	W =  90.000 deg,	P =   0.000 deg,	R =   90.000 deg
};
P[1793]{
   GP1:
	UF : 0, UT : 6,		CONFIG : 'N U T, 0, 0, 0',
	X =  121.033  mm,	Y =   -455.775  mm,	Z =   -252.624  mm,
	W =  90.000 deg,	P =   0.000 deg,	R =   90.000 deg
};
P[1794]{
   GP1:
	UF : 0, UT : 6,		CONFIG : 'N U T, 0, 0, 0',
	X =  121.639  mm,	Y =   -456.875  mm,	Z =   -252.453  mm,
	W =  90.000 deg,	P =   0.000 deg,	R =   90.000 deg
};
P[1795]{
   GP1:
	UF : 0, UT : 6,		CONFIG : 'N U T, 0, 0, 0',
	X =  123.724  mm,	Y =   -460.404  mm,	Z =   -252.749  mm,
	W =  90.000 deg,	P =   0.000 deg,	R =   90.000 deg
};
P[1796]{
   GP1:
	UF : 0, UT : 6,		CONFIG : 'N U T, 0, 0, 0',
	X =  126.627  mm,	Y =   -465.516  mm,	Z =   -252.442  mm,
	W =  90.000 deg,	P =   0.000 deg,	R =   90.000 deg
};
P[1797]{
   GP1:
	UF : 0, UT : 6,		CONFIG : 'N U T, 0, 0, 0',
	X =  128.686  mm,	Y =   -468.983  mm,	Z =   -252.799  mm,
	W =  90.000 deg,	P =   0.000 deg,	R =   90.000 deg
};
P[1798]{
   GP1:
	UF : 0, UT : 6,		CONFIG : 'N U T, 0, 0, 0',
	X =  130.202  mm,	Y =   -471.604  mm,	Z =   -252.810  mm,
	W =  90.000 deg,	P =   0.000 deg,	R =   90.000 deg
};
P[1799]{
   GP1:
	UF : 0, UT : 6,		CONFIG : 'N U T, 0, 0, 0',
	X =  130.436  mm,	Y =   -472.132  mm,	Z =   -252.379  mm,
	W =  90.000 deg,	P =   0.000 deg,	R =   90.000 deg
};
P[1800]{
   GP1:
	UF : 0, UT : 6,		CONFIG : 'N U T, 0, 0, 0',
	X =  130.954  mm,	Y =   -472.905  mm,	Z =   -252.816  mm,
	W =  90.000 deg,	P =   0.000 deg,	R =   90.000 deg
};
P[1801]{
   GP1:
	UF : 0, UT : 6,		CONFIG : 'N U T, 0, 0, 0',
	X =  133.177  mm,	Y =   -476.831  mm,	Z =   -252.548  mm,
	W =  90.000 deg,	P =   0.000 deg,	R =   90.000 deg
};
P[1802]{
   GP1:
	UF : 0, UT : 6,		CONFIG : 'N U T, 0, 0, 0',
	X =  133.538  mm,	Y =   -477.462  mm,	Z =   -252.531  mm,
	W =  90.000 deg,	P =   0.000 deg,	R =   90.000 deg
};
P[1803]{
   GP1:
	UF : 0, UT : 6,		CONFIG : 'N U T, 0, 0, 0',
	X =  134.693  mm,	Y =   -479.414  mm,	Z =   -252.701  mm,
	W =  90.000 deg,	P =   0.000 deg,	R =   90.000 deg
};
P[1804]{
   GP1:
	UF : 0, UT : 6,		CONFIG : 'N U T, 0, 0, 0',
	X =  135.165  mm,	Y =   -480.194  mm,	Z =   -252.830  mm,
	W =  90.000 deg,	P =   0.000 deg,	R =   90.000 deg
};
P[1805]{
   GP1:
	UF : 0, UT : 6,		CONFIG : 'N U T, 0, 0, 0',
	X =  136.001  mm,	Y =   -481.750  mm,	Z =   -252.452  mm,
	W =  90.000 deg,	P =   0.000 deg,	R =   90.000 deg
};
P[1806]{
   GP1:
	UF : 0, UT : 6,		CONFIG : 'N U T, 0, 0, 0',
	X =  137.192  mm,	Y =   -483.729  mm,	Z =   -252.749  mm,
	W =  90.000 deg,	P =   0.000 deg,	R =   90.000 deg
};
P[1807]{
   GP1:
	UF : 0, UT : 6,		CONFIG : 'N U T, 0, 0, 0',
	X =  137.849  mm,	Y =   -484.896  mm,	Z =   -252.640  mm,
	W =  90.000 deg,	P =   0.000 deg,	R =   90.000 deg
};
P[1808]{
   GP1:
	UF : 0, UT : 6,		CONFIG : 'N U T, 0, 0, 0',
	X =  139.190  mm,	Y =   -487.189  mm,	Z =   -252.746  mm,
	W =  90.000 deg,	P =   0.000 deg,	R =   90.000 deg
};
P[1809]{
   GP1:
	UF : 0, UT : 6,		CONFIG : 'N U T, 0, 0, 0',
	X =  141.251  mm,	Y =   -490.781  mm,	Z =   -252.665  mm,
	W =  90.000 deg,	P =   0.000 deg,	R =   90.000 deg
};
P[1810]{
   GP1:
	UF : 0, UT : 6,		CONFIG : 'N U T, 0, 0, 0',
	X =  141.636  mm,	Y =   -491.445  mm,	Z =   -252.673  mm,
	W =  90.000 deg,	P =   0.000 deg,	R =   90.000 deg
};
P[1811]{
   GP1:
	UF : 0, UT : 6,		CONFIG : 'N U T, 0, 0, 0',
	X =  142.493  mm,	Y =   -492.972  mm,	Z =   -252.521  mm,
	W =  90.000 deg,	P =   0.000 deg,	R =   90.000 deg
};
P[1812]{
   GP1:
	UF : 0, UT : 6,		CONFIG : 'N U T, 0, 0, 0',
	X =  142.853  mm,	Y =   -493.613  mm,	Z =   -252.462  mm,
	W =  90.000 deg,	P =   0.000 deg,	R =   90.000 deg
};
P[1813]{
   GP1:
	UF : 0, UT : 6,		CONFIG : 'N U T, 0, 0, 0',
	X =  143.399  mm,	Y =   -494.516  mm,	Z =   -252.613  mm,
	W =  90.000 deg,	P =   0.000 deg,	R =   90.000 deg
};
P[1814]{
   GP1:
	UF : 0, UT : 6,		CONFIG : 'N U T, 0, 0, 0',
	X =  144.231  mm,	Y =   -495.934  mm,	Z =   -252.696  mm,
	W =  90.000 deg,	P =   0.000 deg,	R =   90.000 deg
};
P[1815]{
   GP1:
	UF : 0, UT : 6,		CONFIG : 'N U T, 0, 0, 0',
	X =  144.802  mm,	Y =   -496.952  mm,	Z =   -252.588  mm,
	W =  90.000 deg,	P =   0.000 deg,	R =   90.000 deg
};
P[1816]{
   GP1:
	UF : 0, UT : 6,		CONFIG : 'N U T, 0, 0, 0',
	X =  145.481  mm,	Y =   -498.169  mm,	Z =   -252.452  mm,
	W =  90.000 deg,	P =   0.000 deg,	R =   90.000 deg
};
P[1817]{
   GP1:
	UF : 0, UT : 6,		CONFIG : 'N U T, 0, 0, 0',
	X =  146.292  mm,	Y =   -499.476  mm,	Z =   -252.791  mm,
	W =  90.000 deg,	P =   0.000 deg,	R =   90.000 deg
};
P[1818]{
   GP1:
	UF : 0, UT : 6,		CONFIG : 'N U T, 0, 0, 0',
	X =  146.739  mm,	Y =   -500.274  mm,	Z =   -252.706  mm,
	W =  90.000 deg,	P =   0.000 deg,	R =   90.000 deg
};
P[1819]{
   GP1:
	UF : 0, UT : 6,		CONFIG : 'N U T, 0, 0, 0',
	X =  147.563  mm,	Y =   -501.701  mm,	Z =   -252.713  mm,
	W =  90.000 deg,	P =   0.000 deg,	R =   90.000 deg
};
P[1820]{
   GP1:
	UF : 0, UT : 6,		CONFIG : 'N U T, 0, 0, 0',
	X =  148.493  mm,	Y =   -503.314  mm,	Z =   -252.700  mm,
	W =  90.000 deg,	P =   0.000 deg,	R =   90.000 deg
};
P[1821]{
   GP1:
	UF : 0, UT : 6,		CONFIG : 'N U T, 0, 0, 0',
	X =  150.357  mm,	Y =   -506.621  mm,	Z =   -252.426  mm,
	W =  90.000 deg,	P =   0.000 deg,	R =   90.000 deg
};
P[1822]{
   GP1:
	UF : 0, UT : 6,		CONFIG : 'N U T, 0, 0, 0',
	X =  150.746  mm,	Y =   -507.235  mm,	Z =   -252.633  mm,
	W =  90.000 deg,	P =   0.000 deg,	R =   90.000 deg
};
P[1823]{
   GP1:
	UF : 0, UT : 6,		CONFIG : 'N U T, 0, 0, 0',
	X =  151.308  mm,	Y =   -508.160  mm,	Z =   -252.806  mm,
	W =  90.000 deg,	P =   0.000 deg,	R =   90.000 deg
};
P[1824]{
   GP1:
	UF : 0, UT : 6,		CONFIG : 'N U T, 0, 0, 0',
	X =  151.683  mm,	Y =   -508.837  mm,	Z =   -252.707  mm,
	W =  90.000 deg,	P =   0.000 deg,	R =   90.000 deg
};
P[1825]{
   GP1:
	UF : 0, UT : 6,		CONFIG : 'N U T, 0, 0, 0',
	X =  152.311  mm,	Y =   -509.929  mm,	Z =   -252.694  mm,
	W =  90.000 deg,	P =   0.000 deg,	R =   90.000 deg
};
P[1826]{
   GP1:
	UF : 0, UT : 6,		CONFIG : 'N U T, 0, 0, 0',
	X =  153.128  mm,	Y =   -511.311  mm,	Z =   -252.808  mm,
	W =  90.000 deg,	P =   0.000 deg,	R =   90.000 deg
};
P[1827]{
   GP1:
	UF : 0, UT : 6,		CONFIG : 'N U T, 0, 0, 0',
	X =  154.119  mm,	Y =   -513.068  mm,	Z =   -252.664  mm,
	W =  90.000 deg,	P =   0.000 deg,	R =   90.000 deg
};
P[1828]{
   GP1:
	UF : 0, UT : 6,		CONFIG : 'N U T, 0, 0, 0',
	X =  154.577  mm,	Y =   -513.838  mm,	Z =   -252.751  mm,
	W =  90.000 deg,	P =   0.000 deg,	R =   90.000 deg
};
P[1829]{
   GP1:
	UF : 0, UT : 6,		CONFIG : 'N U T, 0, 0, 0',
	X =  155.039  mm,	Y =   -514.717  mm,	Z =   -252.472  mm,
	W =  90.000 deg,	P =   0.000 deg,	R =   90.000 deg
};
P[1830]{
   GP1:
	UF : 0, UT : 6,		CONFIG : 'N U T, 0, 0, 0',
	X =  155.863  mm,	Y =   -516.048  mm,	Z =   -252.802  mm,
	W =  90.000 deg,	P =   0.000 deg,	R =   90.000 deg
};
P[1831]{
   GP1:
	UF : 0, UT : 6,		CONFIG : 'N U T, 0, 0, 0',
	X =  156.629  mm,	Y =   -517.370  mm,	Z =   -252.825  mm,
	W =  90.000 deg,	P =   0.000 deg,	R =   90.000 deg
};
P[1832]{
   GP1:
	UF : 0, UT : 6,		CONFIG : 'N U T, 0, 0, 0',
	X =  157.305  mm,	Y =   -518.557  mm,	Z =   -252.770  mm,
	W =  90.000 deg,	P =   0.000 deg,	R =   90.000 deg
};
P[1833]{
   GP1:
	UF : 0, UT : 6,		CONFIG : 'N U T, 0, 0, 0',
	X =  157.876  mm,	Y =   -519.576  mm,	Z =   -252.661  mm,
	W =  90.000 deg,	P =   0.000 deg,	R =   90.000 deg
};
P[1834]{
   GP1:
	UF : 0, UT : 6,		CONFIG : 'N U T, 0, 0, 0',
	X =  158.508  mm,	Y =   -520.674  mm,	Z =   -252.645  mm,
	W =  90.000 deg,	P =   0.000 deg,	R =   90.000 deg
};
P[1835]{
   GP1:
	UF : 0, UT : 6,		CONFIG : 'N U T, 0, 0, 0',
	X =  159.166  mm,	Y =   -521.778  mm,	Z =   -252.774  mm,
	W =  90.000 deg,	P =   0.000 deg,	R =   90.000 deg
};
P[1836]{
   GP1:
	UF : 0, UT : 6,		CONFIG : 'N U T, 0, 0, 0',
	X =  160.291  mm,	Y =   -523.722  mm,	Z =   -252.795  mm,
	W =  90.000 deg,	P =   0.000 deg,	R =   90.000 deg
};
P[1837]{
   GP1:
	UF : 0, UT : 6,		CONFIG : 'N U T, 0, 0, 0',
	X =  161.266  mm,	Y =   -525.519  mm,	Z =   -252.405  mm,
	W =  90.000 deg,	P =   0.000 deg,	R =   90.000 deg
};
P[1838]{
   GP1:
	UF : 0, UT : 6,		CONFIG : 'N U T, 0, 0, 0',
	X =  161.814  mm,	Y =   -526.350  mm,	Z =   -252.825  mm,
	W =  90.000 deg,	P =   0.000 deg,	R =   90.000 deg
};
P[1839]{
   GP1:
	UF : 0, UT : 6,		CONFIG : 'N U T, 0, 0, 0',
	X =  162.568  mm,	Y =   -527.699  mm,	Z =   -252.671  mm,
	W =  90.000 deg,	P =   0.000 deg,	R =   90.000 deg
};
P[1840]{
   GP1:
	UF : 0, UT : 6,		CONFIG : 'N U T, 0, 0, 0',
	X =  164.174  mm,	Y =   -530.541  mm,	Z =   -252.453  mm,
	W =  90.000 deg,	P =   0.000 deg,	R =   90.000 deg
};
P[1841]{
   GP1:
	UF : 0, UT : 6,		CONFIG : 'N U T, 0, 0, 0',
	X =  164.838  mm,	Y =   -531.586  mm,	Z =   -252.828  mm,
	W =  90.000 deg,	P =   0.000 deg,	R =   90.000 deg
};
P[1842]{
   GP1:
	UF : 0, UT : 6,		CONFIG : 'N U T, 0, 0, 0',
	X =  165.390  mm,	Y =   -532.385  mm,	Z =   -252.752  mm,
	W =  90.000 deg,	P =   0.000 deg,	R =   90.000 deg
};
P[1843]{
   GP1:
	UF : 0, UT : 6,		CONFIG : 'N U T, 0, 0, 0',
	X =  167.108  mm,	Y =   -533.626  mm,	Z =   -252.674  mm,
	W =  90.000 deg,	P =   0.000 deg,	R =   90.000 deg
};
P[1844]{
   GP1:
	UF : 0, UT : 6,		CONFIG : 'N U T, 0, 0, 0',
	X =  169.365  mm,	Y =   -533.792  mm,	Z =   -252.630  mm,
	W =  90.000 deg,	P =   0.000 deg,	R =   90.000 deg
};
P[1845]{
   GP1:
	UF : 0, UT : 6,		CONFIG : 'N U T, 0, 0, 0',
	X =  171.435  mm,	Y =   -532.869  mm,	Z =   -252.655  mm,
	W =  90.000 deg,	P =   0.000 deg,	R =   90.000 deg
};
P[1846]{
   GP1:
	UF : 0, UT : 6,		CONFIG : 'N U T, 0, 0, 0',
	X =  173.601  mm,	Y =   -531.593  mm,	Z =   -252.810  mm,
	W =  90.000 deg,	P =   0.000 deg,	R =   90.000 deg
};
P[1847]{
   GP1:
	UF : 0, UT : 6,		CONFIG : 'N U T, 0, 0, 0',
	X =  175.185  mm,	Y =   -530.681  mm,	Z =   -252.802  mm,
	W =  90.000 deg,	P =   0.000 deg,	R =   90.000 deg
};
P[1848]{
   GP1:
	UF : 0, UT : 6,		CONFIG : 'N U T, 0, 0, 0',
	X =  175.965  mm,	Y =   -530.243  mm,	Z =   -252.720  mm,
	W =  90.000 deg,	P =   0.000 deg,	R =   90.000 deg
};
P[1849]{
   GP1:
	UF : 0, UT : 6,		CONFIG : 'N U T, 0, 0, 0',
	X =  178.959  mm,	Y =   -528.516  mm,	Z =   -252.708  mm,
	W =  90.000 deg,	P =   0.000 deg,	R =   90.000 deg
};
P[1850]{
   GP1:
	UF : 0, UT : 6,		CONFIG : 'N U T, 0, 0, 0',
	X =  179.592  mm,	Y =   -528.151  mm,	Z =   -252.706  mm,
	W =  90.000 deg,	P =   0.000 deg,	R =   90.000 deg
};
P[1851]{
   GP1:
	UF : 0, UT : 6,		CONFIG : 'N U T, 0, 0, 0',
	X =  180.571  mm,	Y =   -527.618  mm,	Z =   -252.501  mm,
	W =  90.000 deg,	P =   0.000 deg,	R =   90.000 deg
};
P[1852]{
   GP1:
	UF : 0, UT : 6,		CONFIG : 'N U T, 0, 0, 0',
	X =  182.092  mm,	Y =   -526.698  mm,	Z =   -252.768  mm,
	W =  90.000 deg,	P =   0.000 deg,	R =   90.000 deg
};
P[1853]{
   GP1:
	UF : 0, UT : 6,		CONFIG : 'N U T, 0, 0, 0',
	X =  183.945  mm,	Y =   -525.646  mm,	Z =   -252.650  mm,
	W =  90.000 deg,	P =   0.000 deg,	R =   90.000 deg
};
P[1854]{
   GP1:
	UF : 0, UT : 6,		CONFIG : 'N U T, 0, 0, 0',
	X =  184.968  mm,	Y =   -525.038  mm,	Z =   -252.757  mm,
	W =  90.000 deg,	P =   0.000 deg,	R =   90.000 deg
};
P[1855]{
   GP1:
	UF : 0, UT : 6,		CONFIG : 'N U T, 0, 0, 0',
	X =  185.590  mm,	Y =   -524.689  mm,	Z =   -252.697  mm,
	W =  90.000 deg,	P =   0.000 deg,	R =   90.000 deg
};
P[1856]{
   GP1:
	UF : 0, UT : 6,		CONFIG : 'N U T, 0, 0, 0',
	X =  186.996  mm,	Y =   -523.876  mm,	Z =   -252.705  mm,
	W =  90.000 deg,	P =   0.000 deg,	R =   90.000 deg
};
P[1857]{
   GP1:
	UF : 0, UT : 6,		CONFIG : 'N U T, 0, 0, 0',
	X =  188.035  mm,	Y =   -523.275  mm,	Z =   -252.712  mm,
	W =  90.000 deg,	P =   0.000 deg,	R =   90.000 deg
};
P[1858]{
   GP1:
	UF : 0, UT : 6,		CONFIG : 'N U T, 0, 0, 0',
	X =  190.067  mm,	Y =   -522.139  mm,	Z =   -252.484  mm,
	W =  90.000 deg,	P =   0.000 deg,	R =   90.000 deg
};
P[1859]{
   GP1:
	UF : 0, UT : 6,		CONFIG : 'N U T, 0, 0, 0',
	X =  191.179  mm,	Y =   -521.447  mm,	Z =   -252.787  mm,
	W =  90.000 deg,	P =   0.000 deg,	R =   90.000 deg
};
P[1860]{
   GP1:
	UF : 0, UT : 6,		CONFIG : 'N U T, 0, 0, 0',
	X =  192.467  mm,	Y =   -520.771  mm,	Z =   -252.372  mm,
	W =  90.000 deg,	P =   0.000 deg,	R =   90.000 deg
};
P[1861]{
   GP1:
	UF : 0, UT : 6,		CONFIG : 'N U T, 0, 0, 0',
	X =  193.287  mm,	Y =   -520.265  mm,	Z =   -252.573  mm,
	W =  90.000 deg,	P =   0.000 deg,	R =   90.000 deg
};
P[1862]{
   GP1:
	UF : 0, UT : 6,		CONFIG : 'N U T, 0, 0, 0',
	X =  194.439  mm,	Y =   -519.593  mm,	Z =   -252.615  mm,
	W =  90.000 deg,	P =   0.000 deg,	R =   90.000 deg
};
P[1863]{
   GP1:
	UF : 0, UT : 6,		CONFIG : 'N U T, 0, 0, 0',
	X =  195.948  mm,	Y =   -518.720  mm,	Z =   -252.623  mm,
	W =  90.000 deg,	P =   0.000 deg,	R =   90.000 deg
};
P[1864]{
   GP1:
	UF : 0, UT : 6,		CONFIG : 'N U T, 0, 0, 0',
	X =  197.493  mm,	Y =   -517.830  mm,	Z =   -252.617  mm,
	W =  90.000 deg,	P =   0.000 deg,	R =   90.000 deg
};
P[1865]{
   GP1:
	UF : 0, UT : 6,		CONFIG : 'N U T, 0, 0, 0',
	X =  200.110  mm,	Y =   -516.328  mm,	Z =   -252.555  mm,
	W =  90.000 deg,	P =   0.000 deg,	R =   90.000 deg
};
P[1866]{
   GP1:
	UF : 0, UT : 6,		CONFIG : 'N U T, 0, 0, 0',
	X =  201.643  mm,	Y =   -515.402  mm,	Z =   -252.810  mm,
	W =  90.000 deg,	P =   0.000 deg,	R =   90.000 deg
};
P[1867]{
   GP1:
	UF : 0, UT : 6,		CONFIG : 'N U T, 0, 0, 0',
	X =  204.102  mm,	Y =   -514.014  mm,	Z =   -252.615  mm,
	W =  90.000 deg,	P =   0.000 deg,	R =   90.000 deg
};
P[1868]{
   GP1:
	UF : 0, UT : 6,		CONFIG : 'N U T, 0, 0, 0',
	X =  207.922  mm,	Y =   -511.774  mm,	Z =   -252.826  mm,
	W =  90.000 deg,	P =   0.000 deg,	R =   90.000 deg
};
P[1869]{
   GP1:
	UF : 0, UT : 6,		CONFIG : 'N U T, 0, 0, 0',
	X =  208.951  mm,	Y =   -511.199  mm,	Z =   -252.705  mm,
	W =  90.000 deg,	P =   0.000 deg,	R =   90.000 deg
};
P[1870]{
   GP1:
	UF : 0, UT : 6,		CONFIG : 'N U T, 0, 0, 0',
	X =  209.715  mm,	Y =   -510.805  mm,	Z =   -252.417  mm,
	W =  90.000 deg,	P =   0.000 deg,	R =   90.000 deg
};
P[1871]{
   GP1:
	UF : 0, UT : 6,		CONFIG : 'N U T, 0, 0, 0',
	X =  211.770  mm,	Y =   -509.568  mm,	Z =   -252.728  mm,
	W =  90.000 deg,	P =   0.000 deg,	R =   90.000 deg
};
P[1872]{
   GP1:
	UF : 0, UT : 6,		CONFIG : 'N U T, 0, 0, 0',
	X =  213.698  mm,	Y =   -508.504  mm,	Z =   -252.426  mm,
	W =  90.000 deg,	P =   0.000 deg,	R =   90.000 deg
};
P[1873]{
   GP1:
	UF : 0, UT : 6,		CONFIG : 'N U T, 0, 0, 0',
	X =  214.327  mm,	Y =   -508.134  mm,	Z =   -252.466  mm,
	W =  90.000 deg,	P =   0.000 deg,	R =   90.000 deg
};
P[1874]{
   GP1:
	UF : 0, UT : 6,		CONFIG : 'N U T, 0, 0, 0',
	X =  216.740  mm,	Y =   -506.698  mm,	Z =   -252.731  mm,
	W =  90.000 deg,	P =   0.000 deg,	R =   90.000 deg
};
P[1875]{
   GP1:
	UF : 0, UT : 6,		CONFIG : 'N U T, 0, 0, 0',
	X =  218.664  mm,	Y =   -505.597  mm,	Z =   -252.665  mm,
	W =  90.000 deg,	P =   0.000 deg,	R =   90.000 deg
};
P[1876]{
   GP1:
	UF : 0, UT : 6,		CONFIG : 'N U T, 0, 0, 0',
	X =  219.225  mm,	Y =   -505.269  mm,	Z =   -252.692  mm,
	W =  90.000 deg,	P =   0.000 deg,	R =   90.000 deg
};
P[1877]{
   GP1:
	UF : 0, UT : 6,		CONFIG : 'N U T, 0, 0, 0',
	X =  219.970  mm,	Y =   -504.835  mm,	Z =   -252.720  mm,
	W =  90.000 deg,	P =   0.000 deg,	R =   90.000 deg
};
P[1878]{
   GP1:
	UF : 0, UT : 6,		CONFIG : 'N U T, 0, 0, 0',
	X =  220.962  mm,	Y =   -504.250  mm,	Z =   -252.791  mm,
	W =  90.000 deg,	P =   0.000 deg,	R =   90.000 deg
};
P[1879]{
   GP1:
	UF : 0, UT : 6,		CONFIG : 'N U T, 0, 0, 0',
	X =  221.630  mm,	Y =   -503.902  mm,	Z =   -252.565  mm,
	W =  90.000 deg,	P =   0.000 deg,	R =   90.000 deg
};
P[1880]{
   GP1:
	UF : 0, UT : 6,		CONFIG : 'N U T, 0, 0, 0',
	X =  224.735  mm,	Y =   -502.112  mm,	Z =   -252.547  mm,
	W =  90.000 deg,	P =   0.000 deg,	R =   90.000 deg
};
P[1881]{
   GP1:
	UF : 0, UT : 6,		CONFIG : 'N U T, 0, 0, 0',
	X =  226.142  mm,	Y =   -501.253  mm,	Z =   -252.830  mm,
	W =  90.000 deg,	P =   0.000 deg,	R =   90.000 deg
};
P[1882]{
   GP1:
	UF : 0, UT : 6,		CONFIG : 'N U T, 0, 0, 0',
	X =  226.791  mm,	Y =   -500.881  mm,	Z =   -252.815  mm,
	W =  90.000 deg,	P =   0.000 deg,	R =   90.000 deg
};
P[1883]{
   GP1:
	UF : 0, UT : 6,		CONFIG : 'N U T, 0, 0, 0',
	X =  229.123  mm,	Y =   -499.597  mm,	Z =   -252.432  mm,
	W =  90.000 deg,	P =   0.000 deg,	R =   90.000 deg
};
P[1884]{
   GP1:
	UF : 0, UT : 6,		CONFIG : 'N U T, 0, 0, 0',
	X =  232.020  mm,	Y =   -497.862  mm,	Z =   -252.812  mm,
	W =  90.000 deg,	P =   0.000 deg,	R =   90.000 deg
};
P[1885]{
   GP1:
	UF : 0, UT : 6,		CONFIG : 'N U T, 0, 0, 0',
	X =  233.818  mm,	Y =   -496.878  mm,	Z =   -252.480  mm,
	W =  90.000 deg,	P =   0.000 deg,	R =   90.000 deg
};
P[1886]{
   GP1:
	UF : 0, UT : 6,		CONFIG : 'N U T, 0, 0, 0',
	X =  235.203  mm,	Y =   -496.054  mm,	Z =   -252.634  mm,
	W =  90.000 deg,	P =   0.000 deg,	R =   90.000 deg
};
P[1887]{
   GP1:
	UF : 0, UT : 6,		CONFIG : 'N U T, 0, 0, 0',
	X =  236.741  mm,	Y =   -495.166  mm,	Z =   -252.627  mm,
	W =  90.000 deg,	P =   0.000 deg,	R =   90.000 deg
};
P[1888]{
   GP1:
	UF : 0, UT : 6,		CONFIG : 'N U T, 0, 0, 0',
	X =  238.222  mm,	Y =   -494.279  mm,	Z =   -252.825  mm,
	W =  90.000 deg,	P =   0.000 deg,	R =   90.000 deg
};
P[1889]{
   GP1:
	UF : 0, UT : 6,		CONFIG : 'N U T, 0, 0, 0',
	X =  239.025  mm,	Y =   -493.821  mm,	Z =   -252.798  mm,
	W =  90.000 deg,	P =   0.000 deg,	R =   90.000 deg
};
P[1890]{
   GP1:
	UF : 0, UT : 6,		CONFIG : 'N U T, 0, 0, 0',
	X =  241.347  mm,	Y =   -492.505  mm,	Z =   -252.639  mm,
	W =  90.000 deg,	P =   0.000 deg,	R =   90.000 deg
};
P[1891]{
   GP1:
	UF : 0, UT : 6,		CONFIG : 'N U T, 0, 0, 0',
	X =  242.193  mm,	Y =   -492.003  mm,	Z =   -252.724  mm,
	W =  90.000 deg,	P =   0.000 deg,	R =   90.000 deg
};
P[1892]{
   GP1:
	UF : 0, UT : 6,		CONFIG : 'N U T, 0, 0, 0',
	X =  243.870  mm,	Y =   -491.080  mm,	Z =   -252.441  mm,
	W =  90.000 deg,	P =   0.000 deg,	R =   90.000 deg
};
P[1893]{
   GP1:
	UF : 0, UT : 6,		CONFIG : 'N U T, 0, 0, 0',
	X =  245.517  mm,	Y =   -490.107  mm,	Z =   -252.579  mm,
	W =  90.000 deg,	P =   0.000 deg,	R =   90.000 deg
};
P[1894]{
   GP1:
	UF : 0, UT : 6,		CONFIG : 'N U T, 0, 0, 0',
	X =  247.251  mm,	Y =   -489.094  mm,	Z =   -252.653  mm,
	W =  90.000 deg,	P =   0.000 deg,	R =   90.000 deg
};
P[1895]{
   GP1:
	UF : 0, UT : 6,		CONFIG : 'N U T, 0, 0, 0',
	X =  248.017  mm,	Y =   -488.644  mm,	Z =   -252.694  mm,
	W =  90.000 deg,	P =   0.000 deg,	R =   90.000 deg
};
P[1896]{
   GP1:
	UF : 0, UT : 6,		CONFIG : 'N U T, 0, 0, 0',
	X =  250.412  mm,	Y =   -487.278  mm,	Z =   -252.597  mm,
	W =  90.000 deg,	P =   0.000 deg,	R =   90.000 deg
};
P[1897]{
   GP1:
	UF : 0, UT : 6,		CONFIG : 'N U T, 0, 0, 0',
	X =  253.459  mm,	Y =   -485.484  mm,	Z =   -252.810  mm,
	W =  90.000 deg,	P =   0.000 deg,	R =   90.000 deg
};
P[1898]{
   GP1:
	UF : 0, UT : 6,		CONFIG : 'N U T, 0, 0, 0',
	X =  254.839  mm,	Y =   -484.743  mm,	Z =   -252.462  mm,
	W =  90.000 deg,	P =   0.000 deg,	R =   90.000 deg
};
P[1899]{
   GP1:
	UF : 0, UT : 6,		CONFIG : 'N U T, 0, 0, 0',
	X =  256.848  mm,	Y =   -483.527  mm,	Z =   -252.813  mm,
	W =  90.000 deg,	P =   0.000 deg,	R =   90.000 deg
};
P[1900]{
   GP1:
	UF : 0, UT : 6,		CONFIG : 'N U T, 0, 0, 0',
	X =  257.690  mm,	Y =   -483.071  mm,	Z =   -252.619  mm,
	W =  90.000 deg,	P =   0.000 deg,	R =   90.000 deg
};
P[1901]{
   GP1:
	UF : 0, UT : 6,		CONFIG : 'N U T, 0, 0, 0',
	X =  258.224  mm,	Y =   -482.743  mm,	Z =   -252.745  mm,
	W =  90.000 deg,	P =   0.000 deg,	R =   90.000 deg
};
P[1902]{
   GP1:
	UF : 0, UT : 6,		CONFIG : 'N U T, 0, 0, 0',
	X =  259.997  mm,	Y =   -481.774  mm,	Z =   -252.403  mm,
	W =  90.000 deg,	P =   0.000 deg,	R =   90.000 deg
};
P[1903]{
   GP1:
	UF : 0, UT : 6,		CONFIG : 'N U T, 0, 0, 0',
	X =  260.943  mm,	Y =   -481.182  mm,	Z =   -252.691  mm,
	W =  90.000 deg,	P =   0.000 deg,	R =   90.000 deg
};
P[1904]{
   GP1:
	UF : 0, UT : 6,		CONFIG : 'N U T, 0, 0, 0',
	X =  261.562  mm,	Y =   -480.842  mm,	Z =   -252.590  mm,
	W =  90.000 deg,	P =   0.000 deg,	R =   90.000 deg
};
P[1905]{
   GP1:
	UF : 0, UT : 6,		CONFIG : 'N U T, 0, 0, 0',
	X =  262.342  mm,	Y =   -480.409  mm,	Z =   -252.475  mm,
	W =  90.000 deg,	P =   0.000 deg,	R =   90.000 deg
};
P[1906]{
   GP1:
	UF : 0, UT : 6,		CONFIG : 'N U T, 0, 0, 0',
	X =  263.034  mm,	Y =   -480.001  mm,	Z =   -252.532  mm,
	W =  90.000 deg,	P =   0.000 deg,	R =   90.000 deg
};
P[1907]{
   GP1:
	UF : 0, UT : 6,		CONFIG : 'N U T, 0, 0, 0',
	X =  265.284  mm,	Y =   -478.688  mm,	Z =   -252.611  mm,
	W =  90.000 deg,	P =   0.000 deg,	R =   90.000 deg
};
P[1908]{
   GP1:
	UF : 0, UT : 6,		CONFIG : 'N U T, 0, 0, 0',
	X =  266.028  mm,	Y =   -478.230  mm,	Z =   -252.790  mm,
	W =  90.000 deg,	P =   0.000 deg,	R =   90.000 deg
};
P[1909]{
   GP1:
	UF : 0, UT : 6,		CONFIG : 'N U T, 0, 0, 0',
	X =  266.960  mm,	Y =   -477.708  mm,	Z =   -252.694  mm,
	W =  90.000 deg,	P =   0.000 deg,	R =   90.000 deg
};
P[1910]{
   GP1:
	UF : 0, UT : 6,		CONFIG : 'N U T, 0, 0, 0',
	X =  268.343  mm,	Y =   -476.940  mm,	Z =   -252.502  mm,
	W =  90.000 deg,	P =   0.000 deg,	R =   90.000 deg
};
P[1911]{
   GP1:
	UF : 0, UT : 6,		CONFIG : 'N U T, 0, 0, 0',
	X =  269.115  mm,	Y =   -476.487  mm,	Z =   -252.548  mm,
	W =  90.000 deg,	P =   0.000 deg,	R =   90.000 deg
};
P[1912]{
   GP1:
	UF : 0, UT : 6,		CONFIG : 'N U T, 0, 0, 0',
	X =  269.740  mm,	Y =   -476.105  mm,	Z =   -252.679  mm,
	W =  90.000 deg,	P =   0.000 deg,	R =   90.000 deg
};
P[1913]{
   GP1:
	UF : 0, UT : 6,		CONFIG : 'N U T, 0, 0, 0',
	X =  270.986  mm,	Y =   -475.382  mm,	Z =   -252.701  mm,
	W =  90.000 deg,	P =   0.000 deg,	R =   90.000 deg
};
P[1914]{
   GP1:
	UF : 0, UT : 6,		CONFIG : 'N U T, 0, 0, 0',
	X =  273.259  mm,	Y =   -474.061  mm,	Z =   -252.753  mm,
	W =  90.000 deg,	P =   0.000 deg,	R =   90.000 deg
};
P[1915]{
   GP1:
	UF : 0, UT : 6,		CONFIG : 'N U T, 0, 0, 0',
	X =  274.268  mm,	Y =   -473.509  mm,	Z =   -252.561  mm,
	W =  90.000 deg,	P =   0.000 deg,	R =   90.000 deg
};
P[1916]{
   GP1:
	UF : 0, UT : 6,		CONFIG : 'N U T, 0, 0, 0',
	X =  275.028  mm,	Y =   -473.087  mm,	Z =   -252.458  mm,
	W =  90.000 deg,	P =   0.000 deg,	R =   90.000 deg
};
P[1917]{
   GP1:
	UF : 0, UT : 6,		CONFIG : 'N U T, 0, 0, 0',
	X =  276.141  mm,	Y =   -472.401  mm,	Z =   -252.730  mm,
	W =  90.000 deg,	P =   0.000 deg,	R =   90.000 deg
};
P[1918]{
   GP1:
	UF : 0, UT : 6,		CONFIG : 'N U T, 0, 0, 0',
	X =  276.735  mm,	Y =   -472.049  mm,	Z =   -252.779  mm,
	W =  90.000 deg,	P =   0.000 deg,	R =   90.000 deg
};
P[1919]{
   GP1:
	UF : 0, UT : 6,		CONFIG : 'N U T, 0, 0, 0',
	X =  277.424  mm,	Y =   -471.684  mm,	Z =   -252.583  mm,
	W =  90.000 deg,	P =   0.000 deg,	R =   90.000 deg
};
P[1920]{
   GP1:
	UF : 0, UT : 6,		CONFIG : 'N U T, 0, 0, 0',
	X =  282.062  mm,	Y =   -468.993  mm,	Z =   -252.660  mm,
	W =  90.000 deg,	P =   0.000 deg,	R =   90.000 deg
};
P[1921]{
   GP1:
	UF : 0, UT : 6,		CONFIG : 'N U T, 0, 0, 0',
	X =  283.850  mm,	Y =   -467.950  mm,	Z =   -252.730  mm,
	W =  90.000 deg,	P =   0.000 deg,	R =   90.000 deg
};
P[1922]{
   GP1:
	UF : 0, UT : 6,		CONFIG : 'N U T, 0, 0, 0',
	X =  284.704  mm,	Y =   -467.442  mm,	Z =   -252.816  mm,
	W =  90.000 deg,	P =   0.000 deg,	R =   90.000 deg
};
P[1923]{
   GP1:
	UF : 0, UT : 6,		CONFIG : 'N U T, 0, 0, 0',
	X =  286.192  mm,	Y =   -466.605  mm,	Z =   -252.684  mm,
	W =  90.000 deg,	P =   0.000 deg,	R =   90.000 deg
};
P[1924]{
   GP1:
	UF : 0, UT : 6,		CONFIG : 'N U T, 0, 0, 0',
	X =  286.922  mm,	Y =   -466.177  mm,	Z =   -252.723  mm,
	W =  90.000 deg,	P =   0.000 deg,	R =   90.000 deg
};
P[1925]{
   GP1:
	UF : 0, UT : 6,		CONFIG : 'N U T, 0, 0, 0',
	X =  287.987  mm,	Y =   -465.574  mm,	Z =   -252.648  mm,
	W =  90.000 deg,	P =   0.000 deg,	R =   90.000 deg
};
P[1926]{
   GP1:
	UF : 0, UT : 6,		CONFIG : 'N U T, 0, 0, 0',
	X =  288.619  mm,	Y =   -465.211  mm,	Z =   -252.637  mm,
	W =  90.000 deg,	P =   0.000 deg,	R =   90.000 deg
};
P[1927]{
   GP1:
	UF : 0, UT : 6,		CONFIG : 'N U T, 0, 0, 0',
	X =  289.581  mm,	Y =   -464.640  mm,	Z =   -252.733  mm,
	W =  90.000 deg,	P =   0.000 deg,	R =   90.000 deg
};
P[1928]{
   GP1:
	UF : 0, UT : 6,		CONFIG : 'N U T, 0, 0, 0',
	X =  290.356  mm,	Y =   -464.194  mm,	Z =   -252.721  mm,
	W =  90.000 deg,	P =   0.000 deg,	R =   90.000 deg
};
P[1929]{
   GP1:
	UF : 0, UT : 6,		CONFIG : 'N U T, 0, 0, 0',
	X =  292.377  mm,	Y =   -463.040  mm,	Z =   -252.641  mm,
	W =  90.000 deg,	P =   0.000 deg,	R =   90.000 deg
};
P[1930]{
   GP1:
	UF : 0, UT : 6,		CONFIG : 'N U T, 0, 0, 0',
	X =  293.273  mm,	Y =   -462.497  mm,	Z =   -252.801  mm,
	W =  90.000 deg,	P =   0.000 deg,	R =   90.000 deg
};
P[1931]{
   GP1:
	UF : 0, UT : 6,		CONFIG : 'N U T, 0, 0, 0',
	X =  294.470  mm,	Y =   -461.850  mm,	Z =   -252.530  mm,
	W =  90.000 deg,	P =   0.000 deg,	R =   90.000 deg
};
P[1932]{
   GP1:
	UF : 0, UT : 6,		CONFIG : 'N U T, 0, 0, 0',
	X =  295.950  mm,	Y =   -460.990  mm,	Z =   -252.568  mm,
	W =  90.000 deg,	P =   0.000 deg,	R =   90.000 deg
};
P[1933]{
   GP1:
	UF : 0, UT : 6,		CONFIG : 'N U T, 0, 0, 0',
	X =  296.941  mm,	Y =   -460.409  mm,	Z =   -252.612  mm,
	W =  90.000 deg,	P =   0.000 deg,	R =   90.000 deg
};
P[1934]{
   GP1:
	UF : 0, UT : 6,		CONFIG : 'N U T, 0, 0, 0',
	X =  297.549  mm,	Y =   -460.023  mm,	Z =   -252.834  mm,
	W =  90.000 deg,	P =   0.000 deg,	R =   90.000 deg
};
P[1935]{
   GP1:
	UF : 0, UT : 6,		CONFIG : 'N U T, 0, 0, 0',
	X =  299.304  mm,	Y =   -459.025  mm,	Z =   -252.742  mm,
	W =  90.000 deg,	P =   0.000 deg,	R =   90.000 deg
};
P[1936]{
   GP1:
	UF : 0, UT : 6,		CONFIG : 'N U T, 0, 0, 0',
	X =  301.558  mm,	Y =   -457.710  mm,	Z =   -252.816  mm,
	W =  90.000 deg,	P =   0.000 deg,	R =   90.000 deg
};
P[1937]{
   GP1:
	UF : 0, UT : 6,		CONFIG : 'N U T, 0, 0, 0',
	X =  303.096  mm,	Y =   -456.832  mm,	Z =   -252.763  mm,
	W =  90.000 deg,	P =   0.000 deg,	R =   90.000 deg
};
P[1938]{
   GP1:
	UF : 0, UT : 6,		CONFIG : 'N U T, 0, 0, 0',
	X =  304.642  mm,	Y =   -455.947  mm,	Z =   -252.712  mm,
	W =  90.000 deg,	P =   0.000 deg,	R =   90.000 deg
};
P[1939]{
   GP1:
	UF : 0, UT : 6,		CONFIG : 'N U T, 0, 0, 0',
	X =  305.750  mm,	Y =   -455.295  mm,	Z =   -252.786  mm,
	W =  90.000 deg,	P =   0.000 deg,	R =   90.000 deg
};
P[1940]{
   GP1:
	UF : 0, UT : 6,		CONFIG : 'N U T, 0, 0, 0',
	X =  306.856  mm,	Y =   -454.654  mm,	Z =   -252.803  mm,
	W =  90.000 deg,	P =   0.000 deg,	R =   90.000 deg
};
P[1941]{
   GP1:
	UF : 0, UT : 6,		CONFIG : 'N U T, 0, 0, 0',
	X =  307.893  mm,	Y =   -454.128  mm,	Z =   -252.360  mm,
	W =  90.000 deg,	P =   0.000 deg,	R =   90.000 deg
};
P[1942]{
   GP1:
	UF : 0, UT : 6,		CONFIG : 'N U T, 0, 0, 0',
	X =  310.349  mm,	Y =   -452.647  mm,	Z =   -252.746  mm,
	W =  90.000 deg,	P =   0.000 deg,	R =   90.000 deg
};
P[1943]{
   GP1:
	UF : 0, UT : 6,		CONFIG : 'N U T, 0, 0, 0',
	X =  312.349  mm,	Y =   -451.500  mm,	Z =   -252.693  mm,
	W =  90.000 deg,	P =   0.000 deg,	R =   90.000 deg
};
P[1944]{
   GP1:
	UF : 0, UT : 6,		CONFIG : 'N U T, 0, 0, 0',
	X =  315.761  mm,	Y =   -449.533  mm,	Z =   -252.676  mm,
	W =  90.000 deg,	P =   0.000 deg,	R =   90.000 deg
};
P[1945]{
   GP1:
	UF : 0, UT : 6,		CONFIG : 'N U T, 0, 0, 0',
	X =  317.101  mm,	Y =   -448.794  mm,	Z =   -252.463  mm,
	W =  90.000 deg,	P =   0.000 deg,	R =   90.000 deg
};
P[1946]{
   GP1:
	UF : 0, UT : 6,		CONFIG : 'N U T, 0, 0, 0',
	X =  318.080  mm,	Y =   -448.194  mm,	Z =   -252.674  mm,
	W =  90.000 deg,	P =   0.000 deg,	R =   90.000 deg
};
P[1947]{
   GP1:
	UF : 0, UT : 6,		CONFIG : 'N U T, 0, 0, 0',
	X =  320.831  mm,	Y =   -446.598  mm,	Z =   -252.722  mm,
	W =  90.000 deg,	P =   0.000 deg,	R =   90.000 deg
};
P[1948]{
   GP1:
	UF : 0, UT : 6,		CONFIG : 'N U T, 0, 0, 0',
	X =  321.517  mm,	Y =   -446.229  mm,	Z =   -252.556  mm,
	W =  90.000 deg,	P =   0.000 deg,	R =   90.000 deg
};
P[1949]{
   GP1:
	UF : 0, UT : 6,		CONFIG : 'N U T, 0, 0, 0',
	X =  322.230  mm,	Y =   -445.838  mm,	Z =   -252.429  mm,
	W =  90.000 deg,	P =   0.000 deg,	R =   90.000 deg
};
P[1950]{
   GP1:
	UF : 0, UT : 6,		CONFIG : 'N U T, 0, 0, 0',
	X =  322.951  mm,	Y =   -445.377  mm,	Z =   -252.697  mm,
	W =  90.000 deg,	P =   0.000 deg,	R =   90.000 deg
};
P[1951]{
   GP1:
	UF : 0, UT : 6,		CONFIG : 'N U T, 0, 0, 0',
	X =  323.731  mm,	Y =   -444.957  mm,	Z =   -252.518  mm,
	W =  90.000 deg,	P =   0.000 deg,	R =   90.000 deg
};
P[1952]{
   GP1:
	UF : 0, UT : 6,		CONFIG : 'N U T, 0, 0, 0',
	X =  325.935  mm,	Y =   -443.704  mm,	Z =   -252.399  mm,
	W =  90.000 deg,	P =   0.000 deg,	R =   90.000 deg
};
P[1953]{
   GP1:
	UF : 0, UT : 6,		CONFIG : 'N U T, 0, 0, 0',
	X =  327.745  mm,	Y =   -442.608  mm,	Z =   -252.713  mm,
	W =  90.000 deg,	P =   0.000 deg,	R =   90.000 deg
};
P[1954]{
   GP1:
	UF : 0, UT : 6,		CONFIG : 'N U T, 0, 0, 0',
	X =  329.614  mm,	Y =   -441.524  mm,	Z =   -252.739  mm,
	W =  90.000 deg,	P =   0.000 deg,	R =   90.000 deg
};
P[1955]{
   GP1:
	UF : 0, UT : 6,		CONFIG : 'N U T, 0, 0, 0',
	X =  331.082  mm,	Y =   -440.675  mm,	Z =   -252.744  mm,
	W =  90.000 deg,	P =   0.000 deg,	R =   90.000 deg
};
P[1956]{
   GP1:
	UF : 0, UT : 6,		CONFIG : 'N U T, 0, 0, 0',
	X =  334.280  mm,	Y =   -438.871  mm,	Z =   -252.488  mm,
	W =  90.000 deg,	P =   0.000 deg,	R =   90.000 deg
};
P[1957]{
   GP1:
	UF : 0, UT : 6,		CONFIG : 'N U T, 0, 0, 0',
	X =  334.922  mm,	Y =   -438.469  mm,	Z =   -252.683  mm,
	W =  90.000 deg,	P =   0.000 deg,	R =   90.000 deg
};
P[1958]{
   GP1:
	UF : 0, UT : 6,		CONFIG : 'N U T, 0, 0, 0',
	X =  335.829  mm,	Y =   -437.956  mm,	Z =   -252.613  mm,
	W =  90.000 deg,	P =   0.000 deg,	R =   90.000 deg
};
P[1959]{
   GP1:
	UF : 0, UT : 6,		CONFIG : 'N U T, 0, 0, 0',
	X =  341.425  mm,	Y =   -434.760  mm,	Z =   -252.400  mm,
	W =  90.000 deg,	P =   0.000 deg,	R =   90.000 deg
};
P[1960]{
   GP1:
	UF : 0, UT : 6,		CONFIG : 'N U T, 0, 0, 0',
	X =  342.205  mm,	Y =   -434.280  mm,	Z =   -252.582  mm,
	W =  90.000 deg,	P =   0.000 deg,	R =   90.000 deg
};
P[1961]{
   GP1:
	UF : 0, UT : 6,		CONFIG : 'N U T, 0, 0, 0',
	X =  343.140  mm,	Y =   -433.717  mm,	Z =   -252.722  mm,
	W =  90.000 deg,	P =   0.000 deg,	R =   90.000 deg
};
P[1962]{
   GP1:
	UF : 0, UT : 6,		CONFIG : 'N U T, 0, 0, 0',
	X =  344.751  mm,	Y =   -432.816  mm,	Z =   -252.542  mm,
	W =  90.000 deg,	P =   0.000 deg,	R =   90.000 deg
};
P[1963]{
   GP1:
	UF : 0, UT : 6,		CONFIG : 'N U T, 0, 0, 0',
	X =  346.382  mm,	Y =   -431.827  mm,	Z =   -252.832  mm,
	W =  90.000 deg,	P =   0.000 deg,	R =   90.000 deg
};
P[1964]{
   GP1:
	UF : 0, UT : 6,		CONFIG : 'N U T, 0, 0, 0',
	X =  347.688  mm,	Y =   -431.076  mm,	Z =   -252.814  mm,
	W =  90.000 deg,	P =   0.000 deg,	R =   90.000 deg
};
P[1965]{
   GP1:
	UF : 0, UT : 6,		CONFIG : 'N U T, 0, 0, 0',
	X =  348.621  mm,	Y =   -430.536  mm,	Z =   -252.819  mm,
	W =  90.000 deg,	P =   0.000 deg,	R =   90.000 deg
};
P[1966]{
   GP1:
	UF : 0, UT : 6,		CONFIG : 'N U T, 0, 0, 0',
	X =  349.515  mm,	Y =   -430.079  mm,	Z =   -252.454  mm,
	W =  90.000 deg,	P =   0.000 deg,	R =   90.000 deg
};
P[1967]{
   GP1:
	UF : 0, UT : 6,		CONFIG : 'N U T, 0, 0, 0',
	X =  350.430  mm,	Y =   -429.533  mm,	Z =   -252.565  mm,
	W =  90.000 deg,	P =   0.000 deg,	R =   90.000 deg
};
P[1968]{
   GP1:
	UF : 0, UT : 6,		CONFIG : 'N U T, 0, 0, 0',
	X =  352.329  mm,	Y =   -428.432  mm,	Z =   -252.596  mm,
	W =  90.000 deg,	P =   0.000 deg,	R =   90.000 deg
};
P[1969]{
   GP1:
	UF : 0, UT : 6,		CONFIG : 'N U T, 0, 0, 0',
	X =  353.323  mm,	Y =   -427.873  mm,	Z =   -252.503  mm,
	W =  90.000 deg,	P =   0.000 deg,	R =   90.000 deg
};
P[1970]{
   GP1:
	UF : 0, UT : 6,		CONFIG : 'N U T, 0, 0, 0',
	X =  355.225  mm,	Y =   -426.724  mm,	Z =   -252.820  mm,
	W =  90.000 deg,	P =   0.000 deg,	R =   90.000 deg
};
P[1971]{
   GP1:
	UF : 0, UT : 6,		CONFIG : 'N U T, 0, 0, 0',
	X =  356.796  mm,	Y =   -425.864  mm,	Z =   -252.525  mm,
	W =  90.000 deg,	P =   0.000 deg,	R =   90.000 deg
};
P[1972]{
   GP1:
	UF : 0, UT : 6,		CONFIG : 'N U T, 0, 0, 0',
	X =  359.178  mm,	Y =   -424.448  mm,	Z =   -252.776  mm,
	W =  90.000 deg,	P =   0.000 deg,	R =   90.000 deg
};
P[1973]{
   GP1:
	UF : 0, UT : 6,		CONFIG : 'N U T, 0, 0, 0',
	X =  360.047  mm,	Y =   -423.949  mm,	Z =   -252.756  mm,
	W =  90.000 deg,	P =   0.000 deg,	R =   90.000 deg
};
P[1974]{
   GP1:
	UF : 0, UT : 6,		CONFIG : 'N U T, 0, 0, 0',
	X =  362.474  mm,	Y =   -422.565  mm,	Z =   -252.651  mm,
	W =  90.000 deg,	P =   0.000 deg,	R =   90.000 deg
};
P[1975]{
   GP1:
	UF : 0, UT : 6,		CONFIG : 'N U T, 0, 0, 0',
	X =  365.130  mm,	Y =   -421.023  mm,	Z =   -252.708  mm,
	W =  90.000 deg,	P =   0.000 deg,	R =   90.000 deg
};
P[1976]{
   GP1:
	UF : 0, UT : 6,		CONFIG : 'N U T, 0, 0, 0',
	X =  366.227  mm,	Y =   -420.379  mm,	Z =   -252.772  mm,
	W =  90.000 deg,	P =   0.000 deg,	R =   90.000 deg
};
P[1977]{
   GP1:
	UF : 0, UT : 6,		CONFIG : 'N U T, 0, 0, 0',
	X =  367.122  mm,	Y =   -419.802  mm,	Z =   -252.803  mm,
	W =  90.000 deg,	P =   0.000 deg,	R =   90.000 deg
};
P[1978]{
   GP1:
	UF : 0, UT : 6,		CONFIG : 'N U T, 0, 0, 0',
	X =  368.374  mm,	Y =   -418.575  mm,	Z =   -252.469  mm,
	W =  90.000 deg,	P =   0.000 deg,	R =   90.000 deg
};
P[1979]{
   GP1:
	UF : 0, UT : 6,		CONFIG : 'N U T, 0, 0, 0',
	X =  368.785  mm,	Y =   -417.254  mm,	Z =   -252.809  mm,
	W =  90.000 deg,	P =   0.000 deg,	R =   90.000 deg
};
P[1980]{
   GP1:
	UF : 0, UT : 6,		CONFIG : 'N U T, 0, 0, 0',
	X =  368.360  mm,	Y =   -414.366  mm,	Z =   -252.480  mm,
	W =  90.000 deg,	P =   0.000 deg,	R =   90.000 deg
};
P[1981]{
   GP1:
	UF : 0, UT : 6,		CONFIG : 'N U T, 0, 0, 0',
	X =  367.773  mm,	Y =   -413.399  mm,	Z =   -252.657  mm,
	W =  90.000 deg,	P =   0.000 deg,	R =   90.000 deg
};
P[1982]{
   GP1:
	UF : 0, UT : 6,		CONFIG : 'N U T, 0, 0, 0',
	X =  367.339  mm,	Y =   -412.671  mm,	Z =   -252.738  mm,
	W =  90.000 deg,	P =   0.000 deg,	R =   90.000 deg
};
P[1983]{
   GP1:
	UF : 0, UT : 6,		CONFIG : 'N U T, 0, 0, 0',
	X =  366.186  mm,	Y =   -410.633  mm,	Z =   -252.592  mm,
	W =  90.000 deg,	P =   0.000 deg,	R =   90.000 deg
};
P[1984]{
   GP1:
	UF : 0, UT : 6,		CONFIG : 'N U T, 0, 0, 0',
	X =  365.699  mm,	Y =   -409.808  mm,	Z =   -252.659  mm,
	W =  90.000 deg,	P =   0.000 deg,	R =   90.000 deg
};
P[1985]{
   GP1:
	UF : 0, UT : 6,		CONFIG : 'N U T, 0, 0, 0',
	X =  365.311  mm,	Y =   -409.098  mm,	Z =   -252.521  mm,
	W =  90.000 deg,	P =   0.000 deg,	R =   90.000 deg
};
P[1986]{
   GP1:
	UF : 0, UT : 6,		CONFIG : 'N U T, 0, 0, 0',
	X =  364.821  mm,	Y =   -408.260  mm,	Z =   -252.564  mm,
	W =  90.000 deg,	P =   0.000 deg,	R =   90.000 deg
};
P[1987]{
   GP1:
	UF : 0, UT : 6,		CONFIG : 'N U T, 0, 0, 0',
	X =  364.295  mm,	Y =   -407.418  mm,	Z =   -252.808  mm,
	W =  90.000 deg,	P =   0.000 deg,	R =   90.000 deg
};
P[1988]{
   GP1:
	UF : 0, UT : 6,		CONFIG : 'N U T, 0, 0, 0',
	X =  363.207  mm,	Y =   -405.523  mm,	Z =   -252.767  mm,
	W =  90.000 deg,	P =   0.000 deg,	R =   90.000 deg
};
P[1989]{
   GP1:
	UF : 0, UT : 6,		CONFIG : 'N U T, 0, 0, 0',
	X =  362.444  mm,	Y =   -404.155  mm,	Z =   -252.606  mm,
	W =  90.000 deg,	P =   0.000 deg,	R =   90.000 deg
};
P[1990]{
   GP1:
	UF : 0, UT : 6,		CONFIG : 'N U T, 0, 0, 0',
	X =  361.706  mm,	Y =   -402.937  mm,	Z =   -252.815  mm,
	W =  90.000 deg,	P =   0.000 deg,	R =   90.000 deg
};
P[1991]{
   GP1:
	UF : 0, UT : 6,		CONFIG : 'N U T, 0, 0, 0',
	X =  360.656  mm,	Y =   -401.078  mm,	Z =   -252.676  mm,
	W =  90.000 deg,	P =   0.000 deg,	R =   90.000 deg
};
P[1992]{
   GP1:
	UF : 0, UT : 6,		CONFIG : 'N U T, 0, 0, 0',
	X =  360.189  mm,	Y =   -400.292  mm,	Z =   -252.754  mm,
	W =  90.000 deg,	P =   0.000 deg,	R =   90.000 deg
};
P[1993]{
   GP1:
	UF : 0, UT : 6,		CONFIG : 'N U T, 0, 0, 0',
	X =  358.808  mm,	Y =   -397.899  mm,	Z =   -252.748  mm,
	W =  90.000 deg,	P =   0.000 deg,	R =   90.000 deg
};
P[1994]{
   GP1:
	UF : 0, UT : 6,		CONFIG : 'N U T, 0, 0, 0',
	X =  358.417  mm,	Y =   -397.171  mm,	Z =   -252.572  mm,
	W =  90.000 deg,	P =   0.000 deg,	R =   90.000 deg
};
P[1995]{
   GP1:
	UF : 0, UT : 6,		CONFIG : 'N U T, 0, 0, 0',
	X =  356.890  mm,	Y =   -394.545  mm,	Z =   -252.636  mm,
	W =  90.000 deg,	P =   0.000 deg,	R =   90.000 deg
};
P[1996]{
   GP1:
	UF : 0, UT : 6,		CONFIG : 'N U T, 0, 0, 0',
	X =  356.402  mm,	Y =   -393.658  mm,	Z =   -252.493  mm,
	W =  90.000 deg,	P =   0.000 deg,	R =   90.000 deg
};
P[1997]{
   GP1:
	UF : 0, UT : 6,		CONFIG : 'N U T, 0, 0, 0',
	X =  355.249  mm,	Y =   -391.687  mm,	Z =   -252.585  mm,
	W =  90.000 deg,	P =   0.000 deg,	R =   90.000 deg
};
P[1998]{
   GP1:
	UF : 0, UT : 6,		CONFIG : 'N U T, 0, 0, 0',
	X =  354.849  mm,	Y =   -390.997  mm,	Z =   -252.587  mm,
	W =  90.000 deg,	P =   0.000 deg,	R =   90.000 deg
};
P[1999]{
   GP1:
	UF : 0, UT : 6,		CONFIG : 'N U T, 0, 0, 0',
	X =  353.993  mm,	Y =   -389.501  mm,	Z =   -252.539  mm,
	W =  90.000 deg,	P =   0.000 deg,	R =   90.000 deg
};
P[2000]{
   GP1:
	UF : 0, UT : 6,		CONFIG : 'N U T, 0, 0, 0',
	X =  351.343  mm,	Y =   -384.907  mm,	Z =   -252.526  mm,
	W =  90.000 deg,	P =   0.000 deg,	R =   90.000 deg
};
P[2001]{
   GP1:
	UF : 0, UT : 6,		CONFIG : 'N U T, 0, 0, 0',
	X =  350.573  mm,	Y =   -383.591  mm,	Z =   -252.589  mm,
	W =  90.000 deg,	P =   0.000 deg,	R =   90.000 deg
};
P[2002]{
   GP1:
	UF : 0, UT : 6,		CONFIG : 'N U T, 0, 0, 0',
	X =  349.884  mm,	Y =   -382.427  mm,	Z =   -252.693  mm,
	W =  90.000 deg,	P =   0.000 deg,	R =   90.000 deg
};
P[2003]{
   GP1:
	UF : 0, UT : 6,		CONFIG : 'N U T, 0, 0, 0',
	X =  349.052  mm,	Y =   -381.008  mm,	Z =   -252.775  mm,
	W =  90.000 deg,	P =   0.000 deg,	R =   90.000 deg
};
P[2004]{
   GP1:
	UF : 0, UT : 6,		CONFIG : 'N U T, 0, 0, 0',
	X =  348.784  mm,	Y =   -380.450  mm,	Z =   -252.435  mm,
	W =  90.000 deg,	P =   0.000 deg,	R =   90.000 deg
};
P[2005]{
   GP1:
	UF : 0, UT : 6,		CONFIG : 'N U T, 0, 0, 0',
	X =  348.323  mm,	Y =   -379.709  mm,	Z =   -252.641  mm,
	W =  90.000 deg,	P =   0.000 deg,	R =   90.000 deg
};
P[2006]{
   GP1:
	UF : 0, UT : 6,		CONFIG : 'N U T, 0, 0, 0',
	X =  347.762  mm,	Y =   -378.744  mm,	Z =   -252.660  mm,
	W =  90.000 deg,	P =   0.000 deg,	R =   90.000 deg
};
P[2007]{
   GP1:
	UF : 0, UT : 6,		CONFIG : 'N U T, 0, 0, 0',
	X =  345.903  mm,	Y =   -375.503  mm,	Z =   -252.591  mm,
	W =  90.000 deg,	P =   0.000 deg,	R =   90.000 deg
};
P[2008]{
   GP1:
	UF : 0, UT : 6,		CONFIG : 'N U T, 0, 0, 0',
	X =  345.420  mm,	Y =   -374.674  mm,	Z =   -252.615  mm,
	W =  90.000 deg,	P =   0.000 deg,	R =   90.000 deg
};
P[2009]{
   GP1:
	UF : 0, UT : 6,		CONFIG : 'N U T, 0, 0, 0',
	X =  344.910  mm,	Y =   -373.803  mm,	Z =   -252.663  mm,
	W =  90.000 deg,	P =   0.000 deg,	R =   90.000 deg
};
P[2010]{
   GP1:
	UF : 0, UT : 6,		CONFIG : 'N U T, 0, 0, 0',
	X =  343.565  mm,	Y =   -371.489  mm,	Z =   -252.714  mm,
	W =  90.000 deg,	P =   0.000 deg,	R =   90.000 deg
};
P[2011]{
   GP1:
	UF : 0, UT : 6,		CONFIG : 'N U T, 0, 0, 0',
	X =  341.295  mm,	Y =   -367.559  mm,	Z =   -252.718  mm,
	W =  90.000 deg,	P =   0.000 deg,	R =   90.000 deg
};
P[2012]{
   GP1:
	UF : 0, UT : 6,		CONFIG : 'N U T, 0, 0, 0',
	X =  340.901  mm,	Y =   -366.841  mm,	Z =   -252.594  mm,
	W =  90.000 deg,	P =   0.000 deg,	R =   90.000 deg
};
P[2013]{
   GP1:
	UF : 0, UT : 6,		CONFIG : 'N U T, 0, 0, 0',
	X =  339.461  mm,	Y =   -364.415  mm,	Z =   -252.835  mm,
	W =  90.000 deg,	P =   0.000 deg,	R =   90.000 deg
};
P[2014]{
   GP1:
	UF : 0, UT : 6,		CONFIG : 'N U T, 0, 0, 0',
	X =  338.862  mm,	Y =   -363.310  mm,	Z =   -252.595  mm,
	W =  90.000 deg,	P =   0.000 deg,	R =   90.000 deg
};
P[2015]{
   GP1:
	UF : 0, UT : 6,		CONFIG : 'N U T, 0, 0, 0',
	X =  338.044  mm,	Y =   -361.873  mm,	Z =   -252.522  mm,
	W =  90.000 deg,	P =   0.000 deg,	R =   90.000 deg
};
P[2016]{
   GP1:
	UF : 0, UT : 6,		CONFIG : 'N U T, 0, 0, 0',
	X =  337.640  mm,	Y =   -361.200  mm,	Z =   -252.612  mm,
	W =  90.000 deg,	P =   0.000 deg,	R =   90.000 deg
};
P[2017]{
   GP1:
	UF : 0, UT : 6,		CONFIG : 'N U T, 0, 0, 0',
	X =  336.120  mm,	Y =   -358.561  mm,	Z =   -252.590  mm,
	W =  90.000 deg,	P =   0.000 deg,	R =   90.000 deg
};
P[2018]{
   GP1:
	UF : 0, UT : 6,		CONFIG : 'N U T, 0, 0, 0',
	X =  334.606  mm,	Y =   -356.003  mm,	Z =   -252.824  mm,
	W =  90.000 deg,	P =   0.000 deg,	R =   90.000 deg
};
P[2019]{
   GP1:
	UF : 0, UT : 6,		CONFIG : 'N U T, 0, 0, 0',
	X =  334.298  mm,	Y =   -355.404  mm,	Z =   -252.586  mm,
	W =  90.000 deg,	P =   0.000 deg,	R =   90.000 deg
};
P[2020]{
   GP1:
	UF : 0, UT : 6,		CONFIG : 'N U T, 0, 0, 0',
	X =  333.959  mm,	Y =   -354.878  mm,	Z =   -252.807  mm,
	W =  90.000 deg,	P =   0.000 deg,	R =   90.000 deg
};
P[2021]{
   GP1:
	UF : 0, UT : 6,		CONFIG : 'N U T, 0, 0, 0',
	X =  333.431  mm,	Y =   -353.927  mm,	Z =   -252.678  mm,
	W =  90.000 deg,	P =   0.000 deg,	R =   90.000 deg
};
P[2022]{
   GP1:
	UF : 0, UT : 6,		CONFIG : 'N U T, 0, 0, 0',
	X =  331.761  mm,	Y =   -351.041  mm,	Z =   -252.702  mm,
	W =  90.000 deg,	P =   0.000 deg,	R =   90.000 deg
};
P[2023]{
   GP1:
	UF : 0, UT : 6,		CONFIG : 'N U T, 0, 0, 0',
	X =  330.558  mm,	Y =   -348.943  mm,	Z =   -252.646  mm,
	W =  90.000 deg,	P =   0.000 deg,	R =   90.000 deg
};
P[2024]{
   GP1:
	UF : 0, UT : 6,		CONFIG : 'N U T, 0, 0, 0',
	X =  329.988  mm,	Y =   -347.990  mm,	Z =   -252.767  mm,
	W =  90.000 deg,	P =   0.000 deg,	R =   90.000 deg
};
P[2025]{
   GP1:
	UF : 0, UT : 6,		CONFIG : 'N U T, 0, 0, 0',
	X =  328.918  mm,	Y =   -346.033  mm,	Z =   -252.397  mm,
	W =  90.000 deg,	P =   0.000 deg,	R =   90.000 deg
};
P[2026]{
   GP1:
	UF : 0, UT : 6,		CONFIG : 'N U T, 0, 0, 0',
	X =  328.439  mm,	Y =   -345.243  mm,	Z =   -252.541  mm,
	W =  90.000 deg,	P =   0.000 deg,	R =   90.000 deg
};
P[2027]{
   GP1:
	UF : 0, UT : 6,		CONFIG : 'N U T, 0, 0, 0',
	X =  327.923  mm,	Y =   -344.397  mm,	Z =   -252.707  mm,
	W =  90.000 deg,	P =   0.000 deg,	R =   90.000 deg
};
P[2028]{
   GP1:
	UF : 0, UT : 6,		CONFIG : 'N U T, 0, 0, 0',
	X =  327.432  mm,	Y =   -343.560  mm,	Z =   -252.756  mm,
	W =  90.000 deg,	P =   0.000 deg,	R =   90.000 deg
};
P[2029]{
   GP1:
	UF : 0, UT : 6,		CONFIG : 'N U T, 0, 0, 0',
	X =  326.473  mm,	Y =   -341.850  mm,	Z =   -252.582  mm,
	W =  90.000 deg,	P =   0.000 deg,	R =   90.000 deg
};
P[2030]{
   GP1:
	UF : 0, UT : 6,		CONFIG : 'N U T, 0, 0, 0',
	X =  325.689  mm,	Y =   -340.522  mm,	Z =   -252.687  mm,
	W =  90.000 deg,	P =   0.000 deg,	R =   90.000 deg
};
P[2031]{
   GP1:
	UF : 0, UT : 6,		CONFIG : 'N U T, 0, 0, 0',
	X =  325.054  mm,	Y =   -339.439  mm,	Z =   -252.750  mm,
	W =  90.000 deg,	P =   0.000 deg,	R =   90.000 deg
};
P[2032]{
   GP1:
	UF : 0, UT : 6,		CONFIG : 'N U T, 0, 0, 0',
	X =  324.497  mm,	Y =   -338.455  mm,	Z =   -252.679  mm,
	W =  90.000 deg,	P =   0.000 deg,	R =   90.000 deg
};
P[2033]{
   GP1:
	UF : 0, UT : 6,		CONFIG : 'N U T, 0, 0, 0',
	X =  323.302  mm,	Y =   -336.337  mm,	Z =   -252.512  mm,
	W =  90.000 deg,	P =   0.000 deg,	R =   90.000 deg
};
P[2034]{
   GP1:
	UF : 0, UT : 6,		CONFIG : 'N U T, 0, 0, 0',
	X =  322.385  mm,	Y =   -334.826  mm,	Z =   -252.783  mm,
	W =  90.000 deg,	P =   0.000 deg,	R =   90.000 deg
};
P[2035]{
   GP1:
	UF : 0, UT : 6,		CONFIG : 'N U T, 0, 0, 0',
	X =  321.898  mm,	Y =   -333.866  mm,	Z =   -252.375  mm,
	W =  90.000 deg,	P =   0.000 deg,	R =   90.000 deg
};
P[2036]{
   GP1:
	UF : 0, UT : 6,		CONFIG : 'N U T, 0, 0, 0',
	X =  321.440  mm,	Y =   -333.161  mm,	Z =   -252.677  mm,
	W =  90.000 deg,	P =   0.000 deg,	R =   90.000 deg
};
P[2037]{
   GP1:
	UF : 0, UT : 6,		CONFIG : 'N U T, 0, 0, 0',
	X =  320.532  mm,	Y =   -331.536  mm,	Z =   -252.496  mm,
	W =  90.000 deg,	P =   0.000 deg,	R =   90.000 deg
};
P[2038]{
   GP1:
	UF : 0, UT : 6,		CONFIG : 'N U T, 0, 0, 0',
	X =  320.022  mm,	Y =   -330.634  mm,	Z =   -252.432  mm,
	W =  90.000 deg,	P =   0.000 deg,	R =   90.000 deg
};
P[2039]{
   GP1:
	UF : 0, UT : 6,		CONFIG : 'N U T, 0, 0, 0',
	X =  318.655  mm,	Y =   -328.326  mm,	Z =   -252.640  mm,
	W =  90.000 deg,	P =   0.000 deg,	R =   90.000 deg
};
P[2040]{
   GP1:
	UF : 0, UT : 6,		CONFIG : 'N U T, 0, 0, 0',
	X =  317.349  mm,	Y =   -326.016  mm,	Z =   -252.471  mm,
	W =  90.000 deg,	P =   0.000 deg,	R =   90.000 deg
};
P[2041]{
   GP1:
	UF : 0, UT : 6,		CONFIG : 'N U T, 0, 0, 0',
	X =  316.776  mm,	Y =   -325.100  mm,	Z =   -252.740  mm,
	W =  90.000 deg,	P =   0.000 deg,	R =   90.000 deg
};
P[2042]{
   GP1:
	UF : 0, UT : 6,		CONFIG : 'N U T, 0, 0, 0',
	X =  315.397  mm,	Y =   -322.661  mm,	Z =   -252.563  mm,
	W =  90.000 deg,	P =   0.000 deg,	R =   90.000 deg
};
P[2043]{
   GP1:
	UF : 0, UT : 6,		CONFIG : 'N U T, 0, 0, 0',
	X =  314.859  mm,	Y =   -321.752  mm,	Z =   -252.641  mm,
	W =  90.000 deg,	P =   0.000 deg,	R =   90.000 deg
};
P[2044]{
   GP1:
	UF : 0, UT : 6,		CONFIG : 'N U T, 0, 0, 0',
	X =  314.111  mm,	Y =   -320.489  mm,	Z =   -252.762  mm,
	W =  90.000 deg,	P =   0.000 deg,	R =   90.000 deg
};
P[2045]{
   GP1:
	UF : 0, UT : 6,		CONFIG : 'N U T, 0, 0, 0',
	X =  313.561  mm,	Y =   -319.513  mm,	Z =   -252.672  mm,
	W =  90.000 deg,	P =   0.000 deg,	R =   90.000 deg
};
P[2046]{
   GP1:
	UF : 0, UT : 6,		CONFIG : 'N U T, 0, 0, 0',
	X =  312.206  mm,	Y =   -317.108  mm,	Z =   -252.462  mm,
	W =  90.000 deg,	P =   0.000 deg,	R =   90.000 deg
};
P[2047]{
   GP1:
	UF : 0, UT : 6,		CONFIG : 'N U T, 0, 0, 0',
	X =  311.615  mm,	Y =   -316.125  mm,	Z =   -252.616  mm,
	W =  90.000 deg,	P =   0.000 deg,	R =   90.000 deg
};
P[2048]{
   GP1:
	UF : 0, UT : 6,		CONFIG : 'N U T, 0, 0, 0',
	X =  310.423  mm,	Y =   -314.059  mm,	Z =   -252.608  mm,
	W =  90.000 deg,	P =   0.000 deg,	R =   90.000 deg
};
P[2049]{
   GP1:
	UF : 0, UT : 6,		CONFIG : 'N U T, 0, 0, 0',
	X =  309.298  mm,	Y =   -312.149  mm,	Z =   -252.745  mm,
	W =  90.000 deg,	P =   0.000 deg,	R =   90.000 deg
};
P[2050]{
   GP1:
	UF : 0, UT : 6,		CONFIG : 'N U T, 0, 0, 0',
	X =  308.596  mm,	Y =   -310.916  mm,	Z =   -252.679  mm,
	W =  90.000 deg,	P =   0.000 deg,	R =   90.000 deg
};
P[2051]{
   GP1:
	UF : 0, UT : 6,		CONFIG : 'N U T, 0, 0, 0',
	X =  306.728  mm,	Y =   -307.710  mm,	Z =   -252.786  mm,
	W =  90.000 deg,	P =   0.000 deg,	R =   90.000 deg
};
P[2052]{
   GP1:
	UF : 0, UT : 6,		CONFIG : 'N U T, 0, 0, 0',
	X =  306.401  mm,	Y =   -307.042  mm,	Z =   -252.423  mm,
	W =  90.000 deg,	P =   0.000 deg,	R =   90.000 deg
};
P[2053]{
   GP1:
	UF : 0, UT : 6,		CONFIG : 'N U T, 0, 0, 0',
	X =  305.944  mm,	Y =   -306.326  mm,	Z =   -252.692  mm,
	W =  90.000 deg,	P =   0.000 deg,	R =   90.000 deg
};
P[2054]{
   GP1:
	UF : 0, UT : 6,		CONFIG : 'N U T, 0, 0, 0',
	X =  305.128  mm,	Y =   -304.941  mm,	Z =   -252.789  mm,
	W =  90.000 deg,	P =   0.000 deg,	R =   90.000 deg
};
P[2055]{
   GP1:
	UF : 0, UT : 6,		CONFIG : 'N U T, 0, 0, 0',
	X =  304.407  mm,	Y =   -303.658  mm,	Z =   -252.675  mm,
	W =  90.000 deg,	P =   0.000 deg,	R =   90.000 deg
};
P[2056]{
   GP1:
	UF : 0, UT : 6,		CONFIG : 'N U T, 0, 0, 0',
	X =  302.873  mm,	Y =   -300.990  mm,	Z =   -252.631  mm,
	W =  90.000 deg,	P =   0.000 deg,	R =   90.000 deg
};
P[2057]{
   GP1:
	UF : 0, UT : 6,		CONFIG : 'N U T, 0, 0, 0',
	X =  301.802  mm,	Y =   -299.173  mm,	Z =   -252.769  mm,
	W =  90.000 deg,	P =   0.000 deg,	R =   90.000 deg
};
P[2058]{
   GP1:
	UF : 0, UT : 6,		CONFIG : 'N U T, 0, 0, 0',
	X =  301.107  mm,	Y =   -297.950  mm,	Z =   -252.696  mm,
	W =  90.000 deg,	P =   0.000 deg,	R =   90.000 deg
};
P[2059]{
   GP1:
	UF : 0, UT : 6,		CONFIG : 'N U T, 0, 0, 0',
	X =  299.727  mm,	Y =   -295.557  mm,	Z =   -252.689  mm,
	W =  90.000 deg,	P =   0.000 deg,	R =   90.000 deg
};
P[2060]{
   GP1:
	UF : 0, UT : 6,		CONFIG : 'N U T, 0, 0, 0',
	X =  299.064  mm,	Y =   -294.434  mm,	Z =   -252.779  mm,
	W =  90.000 deg,	P =   0.000 deg,	R =   90.000 deg
};
P[2061]{
   GP1:
	UF : 0, UT : 6,		CONFIG : 'N U T, 0, 0, 0',
	X =  298.193  mm,	Y =   -292.918  mm,	Z =   -252.754  mm,
	W =  90.000 deg,	P =   0.000 deg,	R =   90.000 deg
};
P[2062]{
   GP1:
	UF : 0, UT : 6,		CONFIG : 'N U T, 0, 0, 0',
	X =  297.833  mm,	Y =   -292.230  mm,	Z =   -252.523  mm,
	W =  90.000 deg,	P =   0.000 deg,	R =   90.000 deg
};
P[2063]{
   GP1:
	UF : 0, UT : 6,		CONFIG : 'N U T, 0, 0, 0',
	X =  297.470  mm,	Y =   -291.601  mm,	Z =   -252.524  mm,
	W =  90.000 deg,	P =   0.000 deg,	R =   90.000 deg
};
P[2064]{
   GP1:
	UF : 0, UT : 6,		CONFIG : 'N U T, 0, 0, 0',
	X =  296.823  mm,	Y =   -290.497  mm,	Z =   -252.577  mm,
	W =  90.000 deg,	P =   0.000 deg,	R =   90.000 deg
};
P[2065]{
   GP1:
	UF : 0, UT : 6,		CONFIG : 'N U T, 0, 0, 0',
	X =  294.993  mm,	Y =   -287.323  mm,	Z =   -252.560  mm,
	W =  90.000 deg,	P =   0.000 deg,	R =   90.000 deg
};
P[2066]{
   GP1:
	UF : 0, UT : 6,		CONFIG : 'N U T, 0, 0, 0',
	X =  294.531  mm,	Y =   -286.583  mm,	Z =   -252.778  mm,
	W =  90.000 deg,	P =   0.000 deg,	R =   90.000 deg
};
P[2067]{
   GP1:
	UF : 0, UT : 6,		CONFIG : 'N U T, 0, 0, 0',
	X =  293.872  mm,	Y =   -285.426  mm,	Z =   -252.721  mm,
	W =  90.000 deg,	P =   0.000 deg,	R =   90.000 deg
};
P[2068]{
   GP1:
	UF : 0, UT : 6,		CONFIG : 'N U T, 0, 0, 0',
	X =  293.220  mm,	Y =   -284.289  mm,	Z =   -252.690  mm,
	W =  90.000 deg,	P =   0.000 deg,	R =   90.000 deg
};
P[2069]{
   GP1:
	UF : 0, UT : 6,		CONFIG : 'N U T, 0, 0, 0',
	X =  292.644  mm,	Y =   -283.212  mm,	Z =   -252.412  mm,
	W =  90.000 deg,	P =   0.000 deg,	R =   90.000 deg
};
P[2070]{
   GP1:
	UF : 0, UT : 6,		CONFIG : 'N U T, 0, 0, 0',
	X =  291.189  mm,	Y =   -280.785  mm,	Z =   -252.741  mm,
	W =  90.000 deg,	P =   0.000 deg,	R =   90.000 deg
};
P[2071]{
   GP1:
	UF : 0, UT : 6,		CONFIG : 'N U T, 0, 0, 0',
	X =  290.605  mm,	Y =   -279.797  mm,	Z =   -252.827  mm,
	W =  90.000 deg,	P =   0.000 deg,	R =   90.000 deg
};
P[2072]{
   GP1:
	UF : 0, UT : 6,		CONFIG : 'N U T, 0, 0, 0',
	X =  290.103  mm,	Y =   -278.828  mm,	Z =   -252.467  mm,
	W =  90.000 deg,	P =   0.000 deg,	R =   90.000 deg
};
P[2073]{
   GP1:
	UF : 0, UT : 6,		CONFIG : 'N U T, 0, 0, 0',
	X =  289.586  mm,	Y =   -277.988  mm,	Z =   -252.670  mm,
	W =  90.000 deg,	P =   0.000 deg,	R =   90.000 deg
};
P[2074]{
   GP1:
	UF : 0, UT : 6,		CONFIG : 'N U T, 0, 0, 0',
	X =  289.061  mm,	Y =   -277.090  mm,	Z =   -252.707  mm,
	W =  90.000 deg,	P =   0.000 deg,	R =   90.000 deg
};
P[2075]{
   GP1:
	UF : 0, UT : 6,		CONFIG : 'N U T, 0, 0, 0',
	X =  288.227  mm,	Y =   -275.656  mm,	Z =   -252.745  mm,
	W =  90.000 deg,	P =   0.000 deg,	R =   90.000 deg
};
P[2076]{
   GP1:
	UF : 0, UT : 6,		CONFIG : 'N U T, 0, 0, 0',
	X =  286.758  mm,	Y =   -273.133  mm,	Z =   -252.818  mm,
	W =  90.000 deg,	P =   0.000 deg,	R =   90.000 deg
};
P[2077]{
   GP1:
	UF : 0, UT : 6,		CONFIG : 'N U T, 0, 0, 0',
	X =  285.932  mm,	Y =   -271.665  mm,	Z =   -252.690  mm,
	W =  90.000 deg,	P =   0.000 deg,	R =   90.000 deg
};
P[2078]{
   GP1:
	UF : 0, UT : 6,		CONFIG : 'N U T, 0, 0, 0',
	X =  285.487  mm,	Y =   -270.894  mm,	Z =   -252.687  mm,
	W =  90.000 deg,	P =   0.000 deg,	R =   90.000 deg
};
P[2079]{
   GP1:
	UF : 0, UT : 6,		CONFIG : 'N U T, 0, 0, 0',
	X =  284.608  mm,	Y =   -269.358  mm,	Z =   -252.637  mm,
	W =  90.000 deg,	P =   0.000 deg,	R =   90.000 deg
};
P[2080]{
   GP1:
	UF : 0, UT : 6,		CONFIG : 'N U T, 0, 0, 0',
	X =  284.051  mm,	Y =   -268.355  mm,	Z =   -252.505  mm,
	W =  90.000 deg,	P =   0.000 deg,	R =   90.000 deg
};
P[2081]{
   GP1:
	UF : 0, UT : 6,		CONFIG : 'N U T, 0, 0, 0',
	X =  283.691  mm,	Y =   -267.785  mm,	Z =   -252.696  mm,
	W =  90.000 deg,	P =   0.000 deg,	R =   90.000 deg
};
P[2082]{
   GP1:
	UF : 0, UT : 6,		CONFIG : 'N U T, 0, 0, 0',
	X =  283.315  mm,	Y =   -267.122  mm,	Z =   -252.646  mm,
	W =  90.000 deg,	P =   0.000 deg,	R =   90.000 deg
};
P[2083]{
   GP1:
	UF : 0, UT : 6,		CONFIG : 'N U T, 0, 0, 0',
	X =  282.524  mm,	Y =   -265.737  mm,	Z =   -252.597  mm,
	W =  90.000 deg,	P =   0.000 deg,	R =   90.000 deg
};
P[2084]{
   GP1:
	UF : 0, UT : 6,		CONFIG : 'N U T, 0, 0, 0',
	X =  282.041  mm,	Y =   -264.905  mm,	Z =   -252.614  mm,
	W =  90.000 deg,	P =   0.000 deg,	R =   90.000 deg
};
P[2085]{
   GP1:
	UF : 0, UT : 6,		CONFIG : 'N U T, 0, 0, 0',
	X =  281.273  mm,	Y =   -263.611  mm,	Z =   -252.741  mm,
	W =  90.000 deg,	P =   0.000 deg,	R =   90.000 deg
};
P[2086]{
   GP1:
	UF : 0, UT : 6,		CONFIG : 'N U T, 0, 0, 0',
	X =  280.720  mm,	Y =   -262.676  mm,	Z =   -252.826  mm,
	W =  90.000 deg,	P =   0.000 deg,	R =   90.000 deg
};
P[2087]{
   GP1:
	UF : 0, UT : 6,		CONFIG : 'N U T, 0, 0, 0',
	X =  279.498  mm,	Y =   -260.498  mm,	Z =   -252.600  mm,
	W =  90.000 deg,	P =   0.000 deg,	R =   90.000 deg
};
P[2088]{
   GP1:
	UF : 0, UT : 6,		CONFIG : 'N U T, 0, 0, 0',
	X =  278.241  mm,	Y =   -258.307  mm,	Z =   -252.555  mm,
	W =  90.000 deg,	P =   0.000 deg,	R =   90.000 deg
};
P[2089]{
   GP1:
	UF : 0, UT : 6,		CONFIG : 'N U T, 0, 0, 0',
	X =  277.605  mm,	Y =   -257.267  mm,	Z =   -252.772  mm,
	W =  90.000 deg,	P =   0.000 deg,	R =   90.000 deg
};
P[2090]{
   GP1:
	UF : 0, UT : 6,		CONFIG : 'N U T, 0, 0, 0',
	X =  276.606  mm,	Y =   -255.538  mm,	Z =   -252.778  mm,
	W =  90.000 deg,	P =   0.000 deg,	R =   90.000 deg
};
P[2091]{
   GP1:
	UF : 0, UT : 6,		CONFIG : 'N U T, 0, 0, 0',
	X =  276.111  mm,	Y =   -254.684  mm,	Z =   -252.793  mm,
	W =  90.000 deg,	P =   0.000 deg,	R =   90.000 deg
};
P[2092]{
   GP1:
	UF : 0, UT : 6,		CONFIG : 'N U T, 0, 0, 0',
	X =  275.434  mm,	Y =   -253.479  mm,	Z =   -252.672  mm,
	W =  90.000 deg,	P =   0.000 deg,	R =   90.000 deg
};
P[2093]{
   GP1:
	UF : 0, UT : 6,		CONFIG : 'N U T, 0, 0, 0',
	X =  274.084  mm,	Y =   -251.090  mm,	Z =   -252.490  mm,
	W =  90.000 deg,	P =   0.000 deg,	R =   90.000 deg
};
P[2094]{
   GP1:
	UF : 0, UT : 6,		CONFIG : 'N U T, 0, 0, 0',
	X =  273.435  mm,	Y =   -250.006  mm,	Z =   -252.637  mm,
	W =  90.000 deg,	P =   0.000 deg,	R =   90.000 deg
};
P[2095]{
   GP1:
	UF : 0, UT : 6,		CONFIG : 'N U T, 0, 0, 0',
	X =  272.801  mm,	Y =   -248.920  mm,	Z =   -252.673  mm,
	W =  90.000 deg,	P =   0.000 deg,	R =   90.000 deg
};
P[2096]{
   GP1:
	UF : 0, UT : 6,		CONFIG : 'N U T, 0, 0, 0',
	X =  272.408  mm,	Y =   -248.256  mm,	Z =   -252.733  mm,
	W =  90.000 deg,	P =   0.000 deg,	R =   90.000 deg
};
P[2097]{
   GP1:
	UF : 0, UT : 6,		CONFIG : 'N U T, 0, 0, 0',
	X =  271.693  mm,	Y =   -246.951  mm,	Z =   -252.495  mm,
	W =  90.000 deg,	P =   0.000 deg,	R =   90.000 deg
};
P[2098]{
   GP1:
	UF : 0, UT : 6,		CONFIG : 'N U T, 0, 0, 0',
	X =  270.348  mm,	Y =   -244.664  mm,	Z =   -252.646  mm,
	W =  90.000 deg,	P =   0.000 deg,	R =   90.000 deg
};
P[2099]{
   GP1:
	UF : 0, UT : 6,		CONFIG : 'N U T, 0, 0, 0',
	X =  269.751  mm,	Y =   -243.646  mm,	Z =   -252.709  mm,
	W =  90.000 deg,	P =   0.000 deg,	R =   90.000 deg
};
P[2100]{
   GP1:
	UF : 0, UT : 6,		CONFIG : 'N U T, 0, 0, 0',
	X =  269.219  mm,	Y =   -242.756  mm,	Z =   -252.815  mm,
	W =  90.000 deg,	P =   0.000 deg,	R =   90.000 deg
};
P[2101]{
   GP1:
	UF : 0, UT : 6,		CONFIG : 'N U T, 0, 0, 0',
	X =  268.045  mm,	Y =   -240.688  mm,	Z =   -252.692  mm,
	W =  90.000 deg,	P =   0.000 deg,	R =   90.000 deg
};
P[2102]{
   GP1:
	UF : 0, UT : 6,		CONFIG : 'N U T, 0, 0, 0',
	X =  267.626  mm,	Y =   -239.918  mm,	Z =   -252.533  mm,
	W =  90.000 deg,	P =   0.000 deg,	R =   90.000 deg
};
P[2103]{
   GP1:
	UF : 0, UT : 6,		CONFIG : 'N U T, 0, 0, 0',
	X =  267.074  mm,	Y =   -238.958  mm,	Z =   -252.519  mm,
	W =  90.000 deg,	P =   0.000 deg,	R =   90.000 deg
};
P[2104]{
   GP1:
	UF : 0, UT : 6,		CONFIG : 'N U T, 0, 0, 0',
	X =  266.675  mm,	Y =   -238.287  mm,	Z =   -252.597  mm,
	W =  90.000 deg,	P =   0.000 deg,	R =   90.000 deg
};
P[2105]{
   GP1:
	UF : 0, UT : 6,		CONFIG : 'N U T, 0, 0, 0',
	X =  265.932  mm,	Y =   -237.036  mm,	Z =   -252.722  mm,
	W =  90.000 deg,	P =   0.000 deg,	R =   90.000 deg
};
P[2106]{
   GP1:
	UF : 0, UT : 6,		CONFIG : 'N U T, 0, 0, 0',
	X =  265.522  mm,	Y =   -236.346  mm,	Z =   -252.790  mm,
	W =  90.000 deg,	P =   0.000 deg,	R =   90.000 deg
};
P[2107]{
   GP1:
	UF : 0, UT : 6,		CONFIG : 'N U T, 0, 0, 0',
	X =  263.762  mm,	Y =   -233.193  mm,	Z =   -252.419  mm,
	W =  90.000 deg,	P =   0.000 deg,	R =   90.000 deg
};
P[2108]{
   GP1:
	UF : 0, UT : 6,		CONFIG : 'N U T, 0, 0, 0',
	X =  262.690  mm,	Y =   -231.335  mm,	Z =   -252.420  mm,
	W =  90.000 deg,	P =   0.000 deg,	R =   90.000 deg
};
P[2109]{
   GP1:
	UF : 0, UT : 6,		CONFIG : 'N U T, 0, 0, 0',
	X =  261.839  mm,	Y =   -229.923  mm,	Z =   -252.637  mm,
	W =  90.000 deg,	P =   0.000 deg,	R =   90.000 deg
};
P[2110]{
   GP1:
	UF : 0, UT : 6,		CONFIG : 'N U T, 0, 0, 0',
	X =  260.985  mm,	Y =   -228.430  mm,	Z =   -252.583  mm,
	W =  90.000 deg,	P =   0.000 deg,	R =   90.000 deg
};
P[2111]{
   GP1:
	UF : 0, UT : 6,		CONFIG : 'N U T, 0, 0, 0',
	X =  260.190  mm,	Y =   -227.079  mm,	Z =   -252.683  mm,
	W =  90.000 deg,	P =   0.000 deg,	R =   90.000 deg
};
P[2112]{
   GP1:
	UF : 0, UT : 6,		CONFIG : 'N U T, 0, 0, 0',
	X =  259.188  mm,	Y =   -225.326  mm,	Z =   -252.616  mm,
	W =  90.000 deg,	P =   0.000 deg,	R =   90.000 deg
};
P[2113]{
   GP1:
	UF : 0, UT : 6,		CONFIG : 'N U T, 0, 0, 0',
	X =  258.730  mm,	Y =   -224.543  mm,	Z =   -252.646  mm,
	W =  90.000 deg,	P =   0.000 deg,	R =   90.000 deg
};
P[2114]{
   GP1:
	UF : 0, UT : 6,		CONFIG : 'N U T, 0, 0, 0',
	X =  257.586  mm,	Y =   -222.573  mm,	Z =   -252.692  mm,
	W =  90.000 deg,	P =   0.000 deg,	R =   90.000 deg
};
P[2115]{
   GP1:
	UF : 0, UT : 6,		CONFIG : 'N U T, 0, 0, 0',
	X =  256.266  mm,	Y =   -220.216  mm,	Z =   -252.438  mm,
	W =  90.000 deg,	P =   0.000 deg,	R =   90.000 deg
};
P[2116]{
   GP1:
	UF : 0, UT : 6,		CONFIG : 'N U T, 0, 0, 0',
	X =  255.408  mm,	Y =   -218.745  mm,	Z =   -252.495  mm,
	W =  90.000 deg,	P =   0.000 deg,	R =   90.000 deg
};
P[2117]{
   GP1:
	UF : 0, UT : 6,		CONFIG : 'N U T, 0, 0, 0',
	X =  254.538  mm,	Y =   -217.474  mm,	Z =   -252.572  mm,
	W =  90.000 deg,	P =   0.000 deg,	R =   90.000 deg
};
P[2118]{
   GP1:
	UF : 0, UT : 6,		CONFIG : 'N U T, 0, 0, 0',
	X =  253.717  mm,	Y =   -216.791  mm,	Z =   -252.710  mm,
	W =  90.000 deg,	P =   0.000 deg,	R =   90.000 deg
};
P[2119]{
   GP1:
	UF : 0, UT : 6,		CONFIG : 'N U T, 0, 0, 0',
	X =  251.782  mm,	Y =   -216.095  mm,	Z =   -252.512  mm,
	W =  90.000 deg,	P =   0.000 deg,	R =   90.000 deg
};
P[2120]{
   GP1:
	UF : 0, UT : 6,		CONFIG : 'N U T, 0, 0, 0',
	X =  249.609  mm,	Y =   -216.559  mm,	Z =   -252.583  mm,
	W =  90.000 deg,	P =   0.000 deg,	R =   90.000 deg
};
P[2121]{
   GP1:
	UF : 0, UT : 6,		CONFIG : 'N U T, 0, 0, 0',
	X =  247.326  mm,	Y =   -217.841  mm,	Z =   -252.622  mm,
	W =  90.000 deg,	P =   0.000 deg,	R =   90.000 deg
};
P[2122]{
   GP1:
	UF : 0, UT : 6,		CONFIG : 'N U T, 0, 0, 0',
	X =  246.700  mm,	Y =   -218.219  mm,	Z =   -252.722  mm,
	W =  90.000 deg,	P =   0.000 deg,	R =   90.000 deg
};
P[2123]{
   GP1:
	UF : 0, UT : 6,		CONFIG : 'N U T, 0, 0, 0',
	X =  244.571  mm,	Y =   -219.445  mm,	Z =   -252.700  mm,
	W =  90.000 deg,	P =   0.000 deg,	R =   90.000 deg
};
P[2124]{
   GP1:
	UF : 0, UT : 6,		CONFIG : 'N U T, 0, 0, 0',
	X =  243.989  mm,	Y =   -219.793  mm,	Z =   -252.778  mm,
	W =  90.000 deg,	P =   0.000 deg,	R =   90.000 deg
};
P[2125]{
   GP1:
	UF : 0, UT : 6,		CONFIG : 'N U T, 0, 0, 0',
	X =  242.559  mm,	Y =   -220.623  mm,	Z =   -252.806  mm,
	W =  90.000 deg,	P =   0.000 deg,	R =   90.000 deg
};
P[2126]{
   GP1:
	UF : 0, UT : 6,		CONFIG : 'N U T, 0, 0, 0',
	X =  241.395  mm,	Y =   -221.261  mm,	Z =   -252.595  mm,
	W =  90.000 deg,	P =   0.000 deg,	R =   90.000 deg
};
P[2127]{
   GP1:
	UF : 0, UT : 6,		CONFIG : 'N U T, 0, 0, 0',
	X =  240.130  mm,	Y =   -222.005  mm,	Z =   -252.681  mm,
	W =  90.000 deg,	P =   0.000 deg,	R =   90.000 deg
};
P[2128]{
   GP1:
	UF : 0, UT : 6,		CONFIG : 'N U T, 0, 0, 0',
	X =  238.562  mm,	Y =   -222.892  mm,	Z =   -252.562  mm,
	W =  90.000 deg,	P =   0.000 deg,	R =   90.000 deg
};
P[2129]{
   GP1:
	UF : 0, UT : 6,		CONFIG : 'N U T, 0, 0, 0',
	X =  236.502  mm,	Y =   -224.052  mm,	Z =   -252.386  mm,
	W =  90.000 deg,	P =   0.000 deg,	R =   90.000 deg
};
P[2130]{
   GP1:
	UF : 0, UT : 6,		CONFIG : 'N U T, 0, 0, 0',
	X =  236.081  mm,	Y =   -224.367  mm,	Z =   -252.822  mm,
	W =  90.000 deg,	P =   0.000 deg,	R =   90.000 deg
};
P[2131]{
   GP1:
	UF : 0, UT : 6,		CONFIG : 'N U T, 0, 0, 0',
	X =  233.727  mm,	Y =   -225.692  mm,	Z =   -252.612  mm,
	W =  90.000 deg,	P =   0.000 deg,	R =   90.000 deg
};
P[2132]{
   GP1:
	UF : 0, UT : 6,		CONFIG : 'N U T, 0, 0, 0',
	X =  231.279  mm,	Y =   -227.133  mm,	Z =   -252.780  mm,
	W =  90.000 deg,	P =   0.000 deg,	R =   90.000 deg
};
P[2133]{
   GP1:
	UF : 0, UT : 6,		CONFIG : 'N U T, 0, 0, 0',
	X =  229.649  mm,	Y =   -228.038  mm,	Z =   -252.562  mm,
	W =  90.000 deg,	P =   0.000 deg,	R =   90.000 deg
};
P[2134]{
   GP1:
	UF : 0, UT : 6,		CONFIG : 'N U T, 0, 0, 0',
	X =  228.348  mm,	Y =   -228.807  mm,	Z =   -252.672  mm,
	W =  90.000 deg,	P =   0.000 deg,	R =   90.000 deg
};
P[2135]{
   GP1:
	UF : 0, UT : 6,		CONFIG : 'N U T, 0, 0, 0',
	X =  227.528  mm,	Y =   -229.298  mm,	Z =   -252.783  mm,
	W =  90.000 deg,	P =   0.000 deg,	R =   90.000 deg
};
P[2136]{
   GP1:
	UF : 0, UT : 6,		CONFIG : 'N U T, 0, 0, 0',
	X =  226.643  mm,	Y =   -229.796  mm,	Z =   -252.700  mm,
	W =  90.000 deg,	P =   0.000 deg,	R =   90.000 deg
};
P[2137]{
   GP1:
	UF : 0, UT : 6,		CONFIG : 'N U T, 0, 0, 0',
	X =  225.277  mm,	Y =   -230.553  mm,	Z =   -252.501  mm,
	W =  90.000 deg,	P =   0.000 deg,	R =   90.000 deg
};
P[2138]{
   GP1:
	UF : 0, UT : 6,		CONFIG : 'N U T, 0, 0, 0',
	X =  224.488  mm,	Y =   -231.036  mm,	Z =   -252.670  mm,
	W =  90.000 deg,	P =   0.000 deg,	R =   90.000 deg
};
P[2139]{
   GP1:
	UF : 0, UT : 6,		CONFIG : 'N U T, 0, 0, 0',
	X =  222.520  mm,	Y =   -232.152  mm,	Z =   -252.549  mm,
	W =  90.000 deg,	P =   0.000 deg,	R =   90.000 deg
};
P[2140]{
   GP1:
	UF : 0, UT : 6,		CONFIG : 'N U T, 0, 0, 0',
	X =  220.282  mm,	Y =   -233.418  mm,	Z =   -252.387  mm,
	W =  90.000 deg,	P =   0.000 deg,	R =   90.000 deg
};
P[2141]{
   GP1:
	UF : 0, UT : 6,		CONFIG : 'N U T, 0, 0, 0',
	X =  219.312  mm,	Y =   -233.972  mm,	Z =   -252.352  mm,
	W =  90.000 deg,	P =   0.000 deg,	R =   90.000 deg
};
P[2142]{
   GP1:
	UF : 0, UT : 6,		CONFIG : 'N U T, 0, 0, 0',
	X =  218.626  mm,	Y =   -234.442  mm,	Z =   -252.808  mm,
	W =  90.000 deg,	P =   0.000 deg,	R =   90.000 deg
};
P[2143]{
   GP1:
	UF : 0, UT : 6,		CONFIG : 'N U T, 0, 0, 0',
	X =  217.783  mm,	Y =   -234.888  mm,	Z =   -252.552  mm,
	W =  90.000 deg,	P =   0.000 deg,	R =   90.000 deg
};
P[2144]{
   GP1:
	UF : 0, UT : 6,		CONFIG : 'N U T, 0, 0, 0',
	X =  216.136  mm,	Y =   -235.826  mm,	Z =   -252.477  mm,
	W =  90.000 deg,	P =   0.000 deg,	R =   90.000 deg
};
P[2145]{
   GP1:
	UF : 0, UT : 6,		CONFIG : 'N U T, 0, 0, 0',
	X =  215.383  mm,	Y =   -236.318  mm,	Z =   -252.827  mm,
	W =  90.000 deg,	P =   0.000 deg,	R =   90.000 deg
};
P[2146]{
   GP1:
	UF : 0, UT : 6,		CONFIG : 'N U T, 0, 0, 0',
	X =  214.656  mm,	Y =   -236.737  mm,	Z =   -252.821  mm,
	W =  90.000 deg,	P =   0.000 deg,	R =   90.000 deg
};
P[2147]{
   GP1:
	UF : 0, UT : 6,		CONFIG : 'N U T, 0, 0, 0',
	X =  213.209  mm,	Y =   -237.565  mm,	Z =   -252.778  mm,
	W =  90.000 deg,	P =   0.000 deg,	R =   90.000 deg
};
P[2148]{
   GP1:
	UF : 0, UT : 6,		CONFIG : 'N U T, 0, 0, 0',
	X =  212.336  mm,	Y =   -238.048  mm,	Z =   -252.646  mm,
	W =  90.000 deg,	P =   0.000 deg,	R =   90.000 deg
};
P[2149]{
   GP1:
	UF : 0, UT : 6,		CONFIG : 'N U T, 0, 0, 0',
	X =  211.458  mm,	Y =   -238.552  mm,	Z =   -252.629  mm,
	W =  90.000 deg,	P =   0.000 deg,	R =   90.000 deg
};
P[2150]{
   GP1:
	UF : 0, UT : 6,		CONFIG : 'N U T, 0, 0, 0',
	X =  209.386  mm,	Y =   -239.726  mm,	Z =   -252.489  mm,
	W =  90.000 deg,	P =   0.000 deg,	R =   90.000 deg
};
P[2151]{
   GP1:
	UF : 0, UT : 6,		CONFIG : 'N U T, 0, 0, 0',
	X =  205.717  mm,	Y =   -241.859  mm,	Z =   -252.580  mm,
	W =  90.000 deg,	P =   0.000 deg,	R =   90.000 deg
};
P[2152]{
   GP1:
	UF : 0, UT : 6,		CONFIG : 'N U T, 0, 0, 0',
	X =  202.878  mm,	Y =   -243.474  mm,	Z =   -252.429  mm,
	W =  90.000 deg,	P =   0.000 deg,	R =   90.000 deg
};
P[2153]{
   GP1:
	UF : 0, UT : 6,		CONFIG : 'N U T, 0, 0, 0',
	X =  201.978  mm,	Y =   -244.031  mm,	Z =   -252.659  mm,
	W =  90.000 deg,	P =   0.000 deg,	R =   90.000 deg
};
P[2154]{
   GP1:
	UF : 0, UT : 6,		CONFIG : 'N U T, 0, 0, 0',
	X =  200.302  mm,	Y =   -244.992  mm,	Z =   -252.619  mm,
	W =  90.000 deg,	P =   0.000 deg,	R =   90.000 deg
};
P[2155]{
   GP1:
	UF : 0, UT : 6,		CONFIG : 'N U T, 0, 0, 0',
	X =  198.379  mm,	Y =   -246.112  mm,	Z =   -252.679  mm,
	W =  90.000 deg,	P =   0.000 deg,	R =   90.000 deg
};
P[2156]{
   GP1:
	UF : 0, UT : 6,		CONFIG : 'N U T, 0, 0, 0',
	X =  195.518  mm,	Y =   -247.789  mm,	Z =   -252.831  mm,
	W =  90.000 deg,	P =   0.000 deg,	R =   90.000 deg
};
P[2157]{
   GP1:
	UF : 0, UT : 6,		CONFIG : 'N U T, 0, 0, 0',
	X =  188.418  mm,	Y =   -251.888  mm,	Z =   -252.836  mm,
	W =  90.000 deg,	P =   0.000 deg,	R =   90.000 deg
};
P[2158]{
   GP1:
	UF : 0, UT : 6,		CONFIG : 'N U T, 0, 0, 0',
	X =  187.097  mm,	Y =   -252.633  mm,	Z =   -252.722  mm,
	W =  90.000 deg,	P =   0.000 deg,	R =   90.000 deg
};
P[2159]{
   GP1:
	UF : 0, UT : 6,		CONFIG : 'N U T, 0, 0, 0',
	X =  186.203  mm,	Y =   -253.167  mm,	Z =   -252.833  mm,
	W =  90.000 deg,	P =   0.000 deg,	R =   90.000 deg
};
P[2160]{
   GP1:
	UF : 0, UT : 6,		CONFIG : 'N U T, 0, 0, 0',
	X =  184.357  mm,	Y =   -254.176  mm,	Z =   -252.480  mm,
	W =  90.000 deg,	P =   0.000 deg,	R =   90.000 deg
};
P[2161]{
   GP1:
	UF : 0, UT : 6,		CONFIG : 'N U T, 0, 0, 0',
	X =  183.708  mm,	Y =   -254.600  mm,	Z =   -252.787  mm,
	W =  90.000 deg,	P =   0.000 deg,	R =   90.000 deg
};
P[2162]{
   GP1:
	UF : 0, UT : 6,		CONFIG : 'N U T, 0, 0, 0',
	X =  182.473  mm,	Y =   -255.305  mm,	Z =   -252.737  mm,
	W =  90.000 deg,	P =   0.000 deg,	R =   90.000 deg
};
P[2163]{
   GP1:
	UF : 0, UT : 6,		CONFIG : 'N U T, 0, 0, 0',
	X =  177.378  mm,	Y =   -258.199  mm,	Z =   -252.444  mm,
	W =  90.000 deg,	P =   0.000 deg,	R =   90.000 deg
};
P[2164]{
   GP1:
	UF : 0, UT : 6,		CONFIG : 'N U T, 0, 0, 0',
	X =  176.702  mm,	Y =   -258.603  mm,	Z =   -252.520  mm,
	W =  90.000 deg,	P =   0.000 deg,	R =   90.000 deg
};
P[2165]{
   GP1:
	UF : 0, UT : 6,		CONFIG : 'N U T, 0, 0, 0',
	X =  175.885  mm,	Y =   -259.061  mm,	Z =   -252.445  mm,
	W =  90.000 deg,	P =   0.000 deg,	R =   90.000 deg
};
P[2166]{
   GP1:
	UF : 0, UT : 6,		CONFIG : 'N U T, 0, 0, 0',
	X =  174.395  mm,	Y =   -259.957  mm,	Z =   -252.660  mm,
	W =  90.000 deg,	P =   0.000 deg,	R =   90.000 deg
};
P[2167]{
   GP1:
	UF : 0, UT : 6,		CONFIG : 'N U T, 0, 0, 0',
	X =  172.343  mm,	Y =   -261.118  mm,	Z =   -252.517  mm,
	W =  90.000 deg,	P =   0.000 deg,	R =   90.000 deg
};
P[2168]{
   GP1:
	UF : 0, UT : 6,		CONFIG : 'N U T, 0, 0, 0',
	X =  171.309  mm,	Y =   -261.711  mm,	Z =   -252.493  mm,
	W =  90.000 deg,	P =   0.000 deg,	R =   90.000 deg
};
P[2169]{
   GP1:
	UF : 0, UT : 6,		CONFIG : 'N U T, 0, 0, 0',
	X =  169.748  mm,	Y =   -262.641  mm,	Z =   -252.668  mm,
	W =  90.000 deg,	P =   0.000 deg,	R =   90.000 deg
};
P[2170]{
   GP1:
	UF : 0, UT : 6,		CONFIG : 'N U T, 0, 0, 0',
	X =  168.131  mm,	Y =   -263.591  mm,	Z =   -252.766  mm,
	W =  90.000 deg,	P =   0.000 deg,	R =   90.000 deg
};
P[2171]{
   GP1:
	UF : 0, UT : 6,		CONFIG : 'N U T, 0, 0, 0',
	X =  167.485  mm,	Y =   -263.954  mm,	Z =   -252.703  mm,
	W =  90.000 deg,	P =   0.000 deg,	R =   90.000 deg
};
P[2172]{
   GP1:
	UF : 0, UT : 6,		CONFIG : 'N U T, 0, 0, 0',
	X =  166.316  mm,	Y =   -264.619  mm,	Z =   -252.650  mm,
	W =  90.000 deg,	P =   0.000 deg,	R =   90.000 deg
};
P[2173]{
   GP1:
	UF : 0, UT : 6,		CONFIG : 'N U T, 0, 0, 0',
	X =  165.701  mm,	Y =   -264.997  mm,	Z =   -252.785  mm,
	W =  90.000 deg,	P =   0.000 deg,	R =   90.000 deg
};
P[2174]{
   GP1:
	UF : 0, UT : 6,		CONFIG : 'N U T, 0, 0, 0',
	X =  165.047  mm,	Y =   -265.308  mm,	Z =   -252.369  mm,
	W =  90.000 deg,	P =   0.000 deg,	R =   90.000 deg
};
P[2175]{
   GP1:
	UF : 0, UT : 6,		CONFIG : 'N U T, 0, 0, 0',
	X =  163.154  mm,	Y =   -266.397  mm,	Z =   -252.349  mm,
	W =  90.000 deg,	P =   0.000 deg,	R =   90.000 deg
};
P[2176]{
   GP1:
	UF : 0, UT : 6,		CONFIG : 'N U T, 0, 0, 0',
	X =  162.775  mm,	Y =   -266.694  mm,	Z =   -252.835  mm,
	W =  90.000 deg,	P =   0.000 deg,	R =   90.000 deg
};
P[2177]{
   GP1:
	UF : 0, UT : 6,		CONFIG : 'N U T, 0, 0, 0',
	X =  161.593  mm,	Y =   -267.367  mm,	Z =   -252.770  mm,
	W =  90.000 deg,	P =   0.000 deg,	R =   90.000 deg
};
P[2178]{
   GP1:
	UF : 0, UT : 6,		CONFIG : 'N U T, 0, 0, 0',
	X =  160.883  mm,	Y =   -267.766  mm,	Z =   -252.707  mm,
	W =  90.000 deg,	P =   0.000 deg,	R =   90.000 deg
};
P[2179]{
   GP1:
	UF : 0, UT : 6,		CONFIG : 'N U T, 0, 0, 0',
	X =  159.911  mm,	Y =   -268.337  mm,	Z =   -252.768  mm,
	W =  90.000 deg,	P =   0.000 deg,	R =   90.000 deg
};
P[2180]{
   GP1:
	UF : 0, UT : 6,		CONFIG : 'N U T, 0, 0, 0',
	X =  159.193  mm,	Y =   -268.712  mm,	Z =   -252.523  mm,
	W =  90.000 deg,	P =   0.000 deg,	R =   90.000 deg
};
P[2181]{
   GP1:
	UF : 0, UT : 6,		CONFIG : 'N U T, 0, 0, 0',
	X =  157.894  mm,	Y =   -269.494  mm,	Z =   -252.717  mm,
	W =  90.000 deg,	P =   0.000 deg,	R =   90.000 deg
};
P[2182]{
   GP1:
	UF : 0, UT : 6,		CONFIG : 'N U T, 0, 0, 0',
	X =  156.891  mm,	Y =   -270.046  mm,	Z =   -252.548  mm,
	W =  90.000 deg,	P =   0.000 deg,	R =   90.000 deg
};
P[2183]{
   GP1:
	UF : 0, UT : 6,		CONFIG : 'N U T, 0, 0, 0',
	X =  155.213  mm,	Y =   -271.028  mm,	Z =   -252.633  mm,
	W =  90.000 deg,	P =   0.000 deg,	R =   90.000 deg
};
P[2184]{
   GP1:
	UF : 0, UT : 6,		CONFIG : 'N U T, 0, 0, 0',
	X =  154.417  mm,	Y =   -271.451  mm,	Z =   -252.409  mm,
	W =  90.000 deg,	P =   0.000 deg,	R =   90.000 deg
};
P[2185]{
   GP1:
	UF : 0, UT : 6,		CONFIG : 'N U T, 0, 0, 0',
	X =  153.228  mm,	Y =   -272.162  mm,	Z =   -252.561  mm,
	W =  90.000 deg,	P =   0.000 deg,	R =   90.000 deg
};
P[2186]{
   GP1:
	UF : 0, UT : 6,		CONFIG : 'N U T, 0, 0, 0',
	X =  151.384  mm,	Y =   -273.222  mm,	Z =   -252.531  mm,
	W =  90.000 deg,	P =   0.000 deg,	R =   90.000 deg
};
P[2187]{
   GP1:
	UF : 0, UT : 6,		CONFIG : 'N U T, 0, 0, 0',
	X =  128.852  mm,	Y =   -285.383  mm,	Z =   -247.299  mm,
	W =  90.000 deg,	P =   0.000 deg,	R =   90.000 deg
};
P[2188]{
   GP1:
	UF : 0, UT : 6,		CONFIG : 'N U T, 0, 0, 0',
	X =  77.354  mm,	Y =   -315.118  mm,	Z =   -247.299  mm,
	W =  90.000 deg,	P =   0.000 deg,	R =   90.000 deg
};
P[2189]{
   GP1:
	UF : 0, UT : 6,		CONFIG : 'N U T, 0, 0, 0',
	X =  210.000  mm,	Y =   -375.000  mm,	Z =   -250.000  mm,
	W =  90.000 deg,	P =   0.000 deg,	R =   90.000 deg
};
/END
